LIN {X 0,Y 368.084,Z 680.12,A -85,B 0,C 180,E1 -13030.841,E2 -13030.841} C_VEL
LIN {X 0,Y 367.442,Z 693.726,A -85,B 0,C 180,E1 -13031.349,E2 -13031.349} C_VEL
LIN {X 0,Y 366.551,Z 706.591,A -85,B 0,C 180,E1 -13032.062,E2 -13032.062} C_VEL
LIN {X 0,Y 365.621,Z 718.366,A -85,B 0,C 180,E1 -13032.953,E2 -13032.953} C_VEL
LIN {X 0,Y 364.601,Z 729.747,A -85,B 0,C 180,E1 -13034.055,E2 -13034.055} C_VEL
LIN {X 0,Y 363.698,Z 740.032,A -85,B 0,C 180,E1 -13035.309,E2 -13035.309} C_VEL
LIN {X 0,Y 362.713,Z 750.07,A -85,B 0,C 180,E1 -13036.839,E2 -13036.839} C_VEL
LIN {X 0,Y 361.776,Z 758.914,A -85,B 0,C 180,E1 -13038.513,E2 -13038.513} C_VEL
LIN {X 0,Y 361.167,Z 765.962,A -85,B 0,C 180,E1 -13040.195,E2 -13040.195} C_VEL
LIN {X 0,Y 360.675,Z 772.412,A -85,B 0,C 180,E1 -13042.159,E2 -13042.159} C_VEL
LIN {X 0,Y 360.43,Z 776.906,A -85,B 0,C 180,E1 -13043.963,E2 -13043.963} C_VEL
LIN {X 0,Y 360.371,Z 779.772,A -85,B 0,C 180,E1 -13045.524,E2 -13045.524} C_VEL
LIN {X 0,Y 360.303,Z 781.326,A -85,B 0,C 180,E1 -13046.644,E2 -13046.644} C_VEL
LIN {X 0,Y 360.267,Z 782.42,A -85,B 0,C 180,E1 -13047.762,E2 -13047.762} C_VEL
LIN {X 0,Y 360.319,Z 783.103,A -85,B 0,C 180,E1 -13048.881,E2 -13048.881} C_VEL
LIN {X 0,Y 360.36,Z 783.39,A -85,B 0,C 180,E1 -13049.998,E2 -13049.998} C_VEL
LIN {X 0,Y 360.303,Z 783.278,A -85,B 0,C 180,E1 -13051.116,E2 -13051.116} C_VEL
LIN {X 0,Y 360.264,Z 782.727,A -85,B 0,C 180,E1 -13052.234,E2 -13052.234} C_VEL
LIN {X 0,Y 360.301,Z 781.769,A -85,B 0,C 180,E1 -13053.353,E2 -13053.353} C_VEL
LIN {X 0,Y 360.368,Z 780.41,A -85,B 0,C 180,E1 -13054.472,E2 -13054.472} C_VEL
LIN {X 0,Y 360.378,Z 777.924,A -85,B 0,C 180,E1 -13055.959,E2 -13055.959} C_VEL
LIN {X 0,Y 360.68,Z 773.636,A -85,B 0,C 180,E1 -13057.838,E2 -13057.838} C_VEL
LIN {X 0,Y 361.116,Z 768.601,A -85,B 0,C 180,E1 -13059.52,E2 -13059.52} C_VEL
LIN {X 0,Y 361.712,Z 762.283,A -85,B 0,C 180,E1 -13061.202,E2 -13061.202} C_VEL
LIN {X 0,Y 362.686,Z 754.4,A -85,B 0,C 180,E1 -13062.874,E2 -13062.874} C_VEL
LIN {X 0,Y 363.619,Z 746.365,A -85,B 0,C 180,E1 -13064.265,E2 -13064.265} C_VEL
LIN {X 0,Y 364.64,Z 736.582,A -85,B 0,C 180,E1 -13065.653,E2 -13065.653} C_VEL
LIN {X 0,Y 365.815,Z 725.732,A -85,B 0,C 180,E1 -13066.891,E2 -13066.891} C_VEL
LIN {X 0,Y 366.852,Z 715.177,A -85,B 0,C 180,E1 -13067.848,E2 -13067.848} C_VEL
LIN {X 0,Y 367.922,Z 702.54,A -85,B 0,C 180,E1 -13068.731,E2 -13068.731} C_VEL
LIN {X 0,Y 368.816,Z 690.014,A -85,B 0,C 180,E1 -13069.369,E2 -13069.369} C_VEL
LIN {X 0,Y 369.448,Z 677.021,A -85,B 0,C 180,E1 -13069.805,E2 -13069.805} C_VEL
LIN {X 0,Y 370.879,Z 603.724,A -85,B 0,C 180,E1 -13071.351,E2 -13071.351} C_VEL
LIN {X 0,Y 367.392,Z 581.766,A -85,B 0,C 180,E1 -13072.093,E2 -13072.093} C_VEL
LIN {X 0,Y 365.082,Z 570.344,A -85,B 0,C 180,E1 -13072.547,E2 -13072.547} C_VEL
LIN {X 0,Y 366.093,Z 561.386,A -85,B 0,C 180,E1 -13074.677,E2 -13074.677} C_VEL
LIN {X 0,Y 365.722,Z 557.159,A -85,B 0,C 180,E1 -13075.762,E2 -13075.762} C_VEL
LIN {X 0,Y 363.389,Z 545.667,A -85,B 0,C 180,E1 -13078.912,E2 -13078.912} C_VEL
LIN {X 0,Y 361.905,Z 539.407,A -85,B 0,C 180,E1 -13080.781,E2 -13080.781} C_VEL
LIN {X 0,Y 361.851,Z 539.411,A -85,B 0,C 180,E1 -13084.279,E2 -13084.279} C_VEL
LIN {X 0,Y 361.868,Z 539.412,A -85,B 0,C 180,E1 -13087.223,E2 -13087.223} C_VEL
LIN {X 0,Y 361.868,Z 539.412,A -85,B 0,C 180,E1 -13090.761,E2 -13090.761} C_VEL
LIN {X 0,Y 361.817,Z 539.417,A -85,B 0,C 180,E1 -13094.366,E2 -13094.366} C_VEL
LIN {X 0,Y 361.85,Z 539.412,A -85,B 0,C 180,E1 -13097.563,E2 -13097.563} C_VEL
LIN {X 0,Y 361.868,Z 539.408,A -85,B 0,C 180,E1 -13100.971,E2 -13100.971} C_VEL
LIN {X 0,Y 361.867,Z 539.408,A -85,B 0,C 180,E1 -13104.654,E2 -13104.654} C_VEL
LIN {X 0,Y 361.829,Z 539.41,A -85,B 0,C 180,E1 -13108.369,E2 -13108.369} C_VEL
LIN {X 0,Y 361.893,Z 539.406,A -85,B 0,C 180,E1 -13110.954,E2 -13110.954} C_VEL
LIN {X 0,Y 361.945,Z 539.396,A -85,B 0,C 180,E1 -13113.474,E2 -13113.474} C_VEL
LIN {X 0,Y 361.88,Z 539.401,A -85,B 0,C 180,E1 -13117.143,E2 -13117.143} C_VEL
LIN {X 0,Y 361.91,Z 539.394,A -85,B 0,C 180,E1 -13120.723,E2 -13120.723} C_VEL
LIN {X 0,Y 361.936,Z 539.392,A -85,B 0,C 180,E1 -13124.225,E2 -13124.225} C_VEL
LIN {X 0,Y 361.989,Z 539.392,A -85,B 0,C 180,E1 -13126.527,E2 -13126.527} C_VEL
LIN {X 0,Y 362.025,Z 539.389,A -85,B 0,C 180,E1 -13129.937,E2 -13129.937} C_VEL
LIN {X 0,Y 362.14,Z 539.37,A -85,B 0,C 180,E1 -13132.192,E2 -13132.192} C_VEL
LIN {X 0,Y 362.108,Z 539.376,A -85,B 0,C 180,E1 -13134.431,E2 -13134.431} C_VEL
LIN {X 0,Y 362.272,Z 539.356,A -85,B 0,C 180,E1 -13137.776,E2 -13137.776} C_VEL
LIN {X 0,Y 362.418,Z 539.341,A -85,B 0,C 180,E1 -13139.999,E2 -13139.999} C_VEL
LIN {X 0,Y 362.272,Z 539.356,A -85,B 0,C 180,E1 -13142.223,E2 -13142.223} C_VEL
LIN {X 0,Y 362.165,Z 539.372,A -85,B 0,C 180,E1 -13146.686,E2 -13146.686} C_VEL
LIN {X 0,Y 362.063,Z 539.386,A -85,B 0,C 180,E1 -13148.933,E2 -13148.933} C_VEL
LIN {X 0,Y 361.956,Z 539.398,A -85,B 0,C 180,E1 -13152.332,E2 -13152.332} C_VEL
LIN {X 0,Y 361.95,Z 539.401,A -85,B 0,C 180,E1 -13154.62,E2 -13154.62} C_VEL
LIN {X 0,Y 361.943,Z 539.402,A -85,B 0,C 180,E1 -13158.099,E2 -13158.099} C_VEL
LIN {X 0,Y 361.87,Z 539.407,A -85,B 0,C 180,E1 -13161.654,E2 -13161.654} C_VEL
LIN {X 0,Y 361.912,Z 539.488,A -85,B 0,C 180,E1 -13163.307,E2 -13163.307} C_VEL
LIN {X 0,Y 363.986,Z 549.132,A -85,B 0,C 180,E1 -13166.365,E2 -13166.365} C_VEL
LIN {X 0,Y 364.74,Z 552.95,A -85,B 0,C 180,E1 -13167.518,E2 -13167.518} C_VEL
LIN {X 0,Y 367.86,Z 561.593,A -85,B 0,C 180,E1 -13167.947,E2 -13167.947} C_VEL
LIN {X 0,Y 371.419,Z 578.984,A -85,B 0,C 180,E1 -13168.598,E2 -13168.598} C_VEL
LIN {X 0,Y 369.528,Z 660.348,A -85,B 0,C 180,E1 -13170.323,E2 -13170.323} C_VEL
LIN {X 0,Y 368.94,Z 673.355,A -85,B 0,C 180,E1 -13170.816,E2 -13170.816} C_VEL
LIN {X 0,Y 368.184,Z 685.745,A -85,B 0,C 180,E1 -13171.502,E2 -13171.502} C_VEL
LIN {X 0,Y 367.176,Z 697.789,A -85,B 0,C 180,E1 -13172.407,E2 -13172.407} C_VEL
LIN {X 0,Y 366.109,Z 709.182,A -85,B 0,C 180,E1 -13173.514,E2 -13173.514} C_VEL
LIN {X 0,Y 365.054,Z 719.145,A -85,B 0,C 180,E1 -13174.722,E2 -13174.722} C_VEL
LIN {X 0,Y 364.055,Z 727.868,A -85,B 0,C 180,E1 -13176.021,E2 -13176.021} C_VEL
LIN {X 0,Y 363.091,Z 735.885,A -85,B 0,C 180,E1 -13177.48,E2 -13177.48} C_VEL
LIN {X 0,Y 362.237,Z 743.126,A -85,B 0,C 180,E1 -13179.101,E2 -13179.101} C_VEL
LIN {X 0,Y 361.466,Z 749.878,A -85,B 0,C 180,E1 -13181.006,E2 -13181.006} C_VEL
LIN {X 0,Y 360.921,Z 755.115,A -85,B 0,C 180,E1 -13182.963,E2 -13182.963} C_VEL
LIN {X 0,Y 360.596,Z 758.312,A -85,B 0,C 180,E1 -13184.558,E2 -13184.558} C_VEL
LIN {X 0,Y 360.329,Z 760.647,A -85,B 0,C 180,E1 -13186.191,E2 -13186.191} C_VEL
LIN {X 0,Y 360.116,Z 762.378,A -85,B 0,C 180,E1 -13188.432,E2 -13188.432} C_VEL
LIN {X 0,Y 360.063,Z 762.667,A -85,B 0,C 180,E1 -13189.903,E2 -13189.903} C_VEL
LIN {X 0,Y 360.083,Z 762.241,A -85,B 0,C 180,E1 -13191.352,E2 -13191.352} C_VEL
LIN {X 0,Y 360.207,Z 760.809,A -85,B 0,C 180,E1 -13193.124,E2 -13193.124} C_VEL
LIN {X 0,Y 360.484,Z 758.216,A -85,B 0,C 180,E1 -13194.967,E2 -13194.967} C_VEL
LIN {X 0,Y 360.765,Z 754.078,A -85,B 0,C 180,E1 -13196.946,E2 -13196.946} C_VEL
LIN {X 0,Y 361.249,Z 748.549,A -85,B 0,C 180,E1 -13198.87,E2 -13198.87} C_VEL
LIN {X 0,Y 361.869,Z 742.009,A -85,B 0,C 180,E1 -13200.637,E2 -13200.637} C_VEL
LIN {X 0,Y 362.646,Z 734.341,A -85,B 0,C 180,E1 -13202.284,E2 -13202.284} C_VEL
LIN {X 0,Y 363.571,Z 724.85,A -85,B 0,C 180,E1 -13203.913,E2 -13203.913} C_VEL
LIN {X 0,Y 364.526,Z 714.942,A -85,B 0,C 180,E1 -13205.284,E2 -13205.284} C_VEL
LIN {X 0,Y 365.51,Z 704.514,A -85,B 0,C 180,E1 -13206.439,E2 -13206.439} C_VEL
LIN {X 0,Y 366.396,Z 693.123,A -85,B 0,C 180,E1 -13207.443,E2 -13207.443} C_VEL
LIN {X 0,Y 367.292,Z 680.176,A -85,B 0,C 180,E1 -13208.315,E2 -13208.315} C_VEL
LIN {X 0,Y 367.937,Z 667.003,A -85,B 0,C 180,E1 -13208.937,E2 -13208.937} C_VEL
LIN {X 0,Y 368.372,Z 653.798,A -85,B 0,C 180,E1 -13209.333,E2 -13209.333} C_VEL
LIN {X 0,Y 369.729,Z 577.273,A -85,B 0,C 180,E1 -13210.906,E2 -13210.906} C_VEL
LIN {X 0,Y 365.138,Z 554.624,A -85,B 0,C 180,E1 -13211.653,E2 -13211.653} C_VEL
LIN {X 0,Y 364.298,Z 551.805,A -85,B 0,C 180,E1 -13211.782,E2 -13211.782} C_VEL
LIN {X 0,Y 362.153,Z 540.301,A -85,B 0,C 180,E1 -13215.102,E2 -13215.102} C_VEL
LIN {X 0,Y 361.997,Z 539.395,A -85,B 0,C 180,E1 -13215.383,E2 -13215.383} C_VEL
LIN {X 0,Y 361.966,Z 539.4,A -85,B 0,C 180,E1 -13218.806,E2 -13218.806} C_VEL
LIN {X 0,Y 362.118,Z 539.375,A -85,B 0,C 180,E1 -13222.194,E2 -13222.194} C_VEL
LIN {X 0,Y 362.111,Z 539.377,A -85,B 0,C 180,E1 -13224.433,E2 -13224.433} C_VEL
LIN {X 0,Y 362.28,Z 539.354,A -85,B 0,C 180,E1 -13227.778,E2 -13227.778} C_VEL
LIN {X 0,Y 362.425,Z 539.336,A -85,B 0,C 180,E1 -13230.002,E2 -13230.002} C_VEL
LIN {X 0,Y 362.28,Z 539.354,A -85,B 0,C 180,E1 -13232.225,E2 -13232.225} C_VEL
LIN {X 0,Y 362.159,Z 539.372,A -85,B 0,C 180,E1 -13236.688,E2 -13236.688} C_VEL
LIN {X 0,Y 362.103,Z 539.378,A -85,B 0,C 180,E1 -13238.513,E2 -13238.513} C_VEL
LIN {X 0,Y 361.349,Z 539.476,A -85,B 0,C 180,E1 -13239.441,E2 -13239.441} C_VEL
LIN {X 0,Y 358.415,Z 539.841,A -85,B 0,C 180,E1 -13240.948,E2 -13240.948} C_VEL
LIN {X 0,Y 355.996,Z 540.137,A -85,B 0,C 180,E1 -13242.167,E2 -13242.167} C_VEL
LIN {X 0,Y 354.993,Z 540.268,A -85,B 0,C 180,E1 -13243.112,E2 -13243.112} C_VEL
LIN {X 0,Y 354.927,Z 540.269,A -85,B 0,C 180,E1 -13243.431,E2 -13243.431} C_VEL
LIN {X 0,Y 354.898,Z 540.278,A -85,B 0,C 180,E1 -13247.282,E2 -13247.282} C_VEL
LIN {X 0,Y 354.84,Z 540.285,A -85,B 0,C 180,E1 -13250.888,E2 -13250.888} C_VEL
LIN {X 0,Y 354.862,Z 540.279,A -85,B 0,C 180,E1 -13254.578,E2 -13254.578} C_VEL
LIN {X 0,Y 354.882,Z 540.281,A -85,B 0,C 180,E1 -13257.098,E2 -13257.098} C_VEL
LIN {X 0,Y 354.801,Z 540.29,A -85,B 0,C 180,E1 -13261,E2 -13261} C_VEL
LIN {X 0,Y 354.808,Z 540.287,A -85,B 0,C 180,E1 -13263.703,E2 -13263.703} C_VEL
LIN {X 0,Y 354.799,Z 540.286,A -85,B 0,C 180,E1 -13266.461,E2 -13266.461} C_VEL
LIN {X 0,Y 354.826,Z 540.288,A -85,B 0,C 180,E1 -13269.425,E2 -13269.425} C_VEL
LIN {X 0,Y 354.792,Z 540.289,A -85,B 0,C 180,E1 -13272.869,E2 -13272.869} C_VEL
LIN {X 0,Y 354.784,Z 540.288,A -85,B 0,C 180,E1 -13276.107,E2 -13276.107} C_VEL
LIN {X 0,Y 354.791,Z 540.291,A -85,B 0,C 180,E1 -13279.18,E2 -13279.18} C_VEL
LIN {X 0,Y 354.811,Z 540.284,A -85,B 0,C 180,E1 -13282.404,E2 -13282.404} C_VEL
LIN {X 0,Y 354.816,Z 540.285,A -85,B 0,C 180,E1 -13284.942,E2 -13284.942} C_VEL
LIN {X 0,Y 354.797,Z 540.286,A -85,B 0,C 180,E1 -13288.406,E2 -13288.406} C_VEL
LIN {X 0,Y 354.856,Z 540.285,A -85,B 0,C 180,E1 -13291.62,E2 -13291.62} C_VEL
LIN {X 0,Y 354.904,Z 540.274,A -85,B 0,C 180,E1 -13294.174,E2 -13294.174} C_VEL
LIN {X 0,Y 354.823,Z 540.286,A -85,B 0,C 180,E1 -13297.894,E2 -13297.894} C_VEL
LIN {X 0,Y 354.896,Z 540.277,A -85,B 0,C 180,E1 -13301.909,E2 -13301.909} C_VEL
LIN {X 0,Y 354.949,Z 540.271,A -85,B 0,C 180,E1 -13305.982,E2 -13305.982} C_VEL
LIN {X 0,Y 354.984,Z 540.269,A -85,B 0,C 180,E1 -13309.737,E2 -13309.737} C_VEL
LIN {X 0,Y 355.132,Z 540.246,A -85,B 0,C 180,E1 -13313.181,E2 -13313.181} C_VEL
LIN {X 0,Y 355.251,Z 540.235,A -85,B 0,C 180,E1 -13317.733,E2 -13317.733} C_VEL
LIN {X 0,Y 355.403,Z 540.215,A -85,B 0,C 180,E1 -13320.001,E2 -13320.001} C_VEL
LIN {X 0,Y 355.251,Z 540.232,A -85,B 0,C 180,E1 -13322.268,E2 -13322.268} C_VEL
LIN {X 0,Y 355.146,Z 540.243,A -85,B 0,C 180,E1 -13326.82,E2 -13326.82} C_VEL
LIN {X 0,Y 355.023,Z 540.258,A -85,B 0,C 180,E1 -13329.113,E2 -13329.113} C_VEL
LIN {X 0,Y 354.929,Z 540.271,A -85,B 0,C 180,E1 -13332.581,E2 -13332.581} C_VEL
LIN {X 0,Y 354.898,Z 540.279,A -85,B 0,C 180,E1 -13336.096,E2 -13336.096} C_VEL
LIN {X 0,Y 354.912,Z 540.274,A -85,B 0,C 180,E1 -13338.472,E2 -13338.472} C_VEL
LIN {X 0,Y 354.824,Z 540.289,A -85,B 0,C 180,E1 -13342.107,E2 -13342.107} C_VEL
LIN {X 0,Y 354.906,Z 540.276,A -85,B 0,C 180,E1 -13345.827,E2 -13345.827} C_VEL
LIN {X 0,Y 354.826,Z 540.285,A -85,B 0,C 180,E1 -13349.682,E2 -13349.682} C_VEL
LIN {X 0,Y 354.814,Z 540.286,A -85,B 0,C 180,E1 -13353.702,E2 -13353.702} C_VEL
LIN {X 0,Y 354.806,Z 540.289,A -85,B 0,C 180,E1 -13356.459,E2 -13356.459} C_VEL
LIN {X 0,Y 354.832,Z 540.282,A -85,B 0,C 180,E1 -13359.423,E2 -13359.423} C_VEL
LIN {X 0,Y 354.795,Z 540.287,A -85,B 0,C 180,E1 -13362.867,E2 -13362.867} C_VEL
LIN {X 0,Y 354.775,Z 540.293,A -85,B 0,C 180,E1 -13366.103,E2 -13366.103} C_VEL
LIN {X 0,Y 354.796,Z 540.286,A -85,B 0,C 180,E1 -13369.178,E2 -13369.178} C_VEL
LIN {X 0,Y 354.82,Z 540.289,A -85,B 0,C 180,E1 -13372.401,E2 -13372.401} C_VEL
LIN {X 0,Y 354.819,Z 540.285,A -85,B 0,C 180,E1 -13374.94,E2 -13374.94} C_VEL
LIN {X 0,Y 354.801,Z 540.292,A -85,B 0,C 180,E1 -13378.404,E2 -13378.404} C_VEL
LIN {X 0,Y 354.856,Z 540.352,A -85,B 0,C 180,E1 -13380.034,E2 -13380.034} C_VEL
LIN {X 0,Y 357.26,Z 551.762,A -85,B 0,C 180,E1 -13383.097,E2 -13383.097} C_VEL
LIN {X 0,Y 358.602,Z 559.43,A -85,B 0,C 180,E1 -13385.078,E2 -13385.078} C_VEL
LIN {X 0,Y 357.874,Z 568.426,A -85,B 0,C 180,E1 -13387.225,E2 -13387.225} C_VEL
LIN {X 0,Y 357.564,Z 571.17,A -85,B 0,C 180,E1 -13387.87,E2 -13387.87} C_VEL
LIN {X 0,Y 362.726,Z 604.121,A -85,B 0,C 180,E1 -13388.896,E2 -13388.896} C_VEL
LIN {X 0,Y 361.331,Z 679.629,A -85,B 0,C 180,E1 -13390.505,E2 -13390.505} C_VEL
LIN {X 0,Y 360.654,Z 693.32,A -85,B 0,C 180,E1 -13391.022,E2 -13391.022} C_VEL
LIN {X 0,Y 359.796,Z 705.738,A -85,B 0,C 180,E1 -13391.713,E2 -13391.713} C_VEL
LIN {X 0,Y 358.808,Z 717.665,A -85,B 0,C 180,E1 -13392.619,E2 -13392.619} C_VEL
LIN {X 0,Y 357.724,Z 729.14,A -85,B 0,C 180,E1 -13393.741,E2 -13393.741} C_VEL
LIN {X 0,Y 356.804,Z 739.453,A -85,B 0,C 180,E1 -13395.008,E2 -13395.008} C_VEL
LIN {X 0,Y 355.739,Z 749.626,A -85,B 0,C 180,E1 -13396.576,E2 -13396.576} C_VEL
LIN {X 0,Y 354.759,Z 758.519,A -85,B 0,C 180,E1 -13398.283,E2 -13398.283} C_VEL
LIN {X 0,Y 354.129,Z 765.615,A -85,B 0,C 180,E1 -13399.998,E2 -13399.998} C_VEL
LIN {X 0,Y 353.619,Z 772.097,A -85,B 0,C 180,E1 -13402.001,E2 -13402.001} C_VEL
LIN {X 0,Y 353.324,Z 777.005,A -85,B 0,C 180,E1 -13404.022,E2 -13404.022} C_VEL
LIN {X 0,Y 353.284,Z 779.509,A -85,B 0,C 180,E1 -13405.434,E2 -13405.434} C_VEL
LIN {X 0,Y 353.225,Z 781.075,A -85,B 0,C 180,E1 -13406.576,E2 -13406.576} C_VEL
LIN {X 0,Y 353.175,Z 782.189,A -85,B 0,C 180,E1 -13407.717,E2 -13407.717} C_VEL
LIN {X 0,Y 353.219,Z 782.882,A -85,B 0,C 180,E1 -13408.858,E2 -13408.858} C_VEL
LIN {X 0,Y 353.263,Z 783.178,A -85,B 0,C 180,E1 -13409.998,E2 -13409.998} C_VEL
LIN {X 0,Y 353.204,Z 783.078,A -85,B 0,C 180,E1 -13411.139,E2 -13411.139} C_VEL
LIN {X 0,Y 353.173,Z 782.544,A -85,B 0,C 180,E1 -13412.279,E2 -13412.279} C_VEL
LIN {X 0,Y 353.223,Z 781.596,A -85,B 0,C 180,E1 -13413.42,E2 -13413.42} C_VEL
LIN {X 0,Y 353.281,Z 780.249,A -85,B 0,C 180,E1 -13414.562,E2 -13414.562} C_VEL
LIN {X 0,Y 353.297,Z 778.061,A -85,B 0,C 180,E1 -13415.935,E2 -13415.935} C_VEL
LIN {X 0,Y 353.624,Z 773.526,A -85,B 0,C 180,E1 -13417.995,E2 -13417.995} C_VEL
LIN {X 0,Y 354.076,Z 768.515,A -85,B 0,C 180,E1 -13419.711,E2 -13419.711} C_VEL
LIN {X 0,Y 354.713,Z 762.222,A -85,B 0,C 180,E1 -13421.426,E2 -13421.426} C_VEL
LIN {X 0,Y 355.741,Z 754.384,A -85,B 0,C 180,E1 -13423.13,E2 -13423.13} C_VEL
LIN {X 0,Y 356.705,Z 746.384,A -85,B 0,C 180,E1 -13424.547,E2 -13424.547} C_VEL
LIN {X 0,Y 357.795,Z 736.642,A -85,B 0,C 180,E1 -13425.96,E2 -13425.96} C_VEL
LIN {X 0,Y 359.026,Z 725.85,A -85,B 0,C 180,E1 -13427.22,E2 -13427.22} C_VEL
LIN {X 0,Y 360.124,Z 715.408,A -85,B 0,C 180,E1 -13428.193,E2 -13428.193} C_VEL
LIN {X 0,Y 361.232,Z 702.941,A -85,B 0,C 180,E1 -13429.091,E2 -13429.091} C_VEL
LIN {X 0,Y 362.16,Z 690.663,A -85,B 0,C 180,E1 -13429.74,E2 -13429.74} C_VEL
LIN {X 0,Y 362.801,Z 678.427,A -85,B 0,C 180,E1 -13430.183,E2 -13430.183} C_VEL
LIN {X 0,Y 364.355,Z 604.435,A -85,B 0,C 180,E1 -13431.787,E2 -13431.787} C_VEL
LIN {X 0,Y 360.878,Z 582.501,A -85,B 0,C 180,E1 -13432.549,E2 -13432.549} C_VEL
LIN {X 0,Y 358.355,Z 570.184,A -85,B 0,C 180,E1 -13433.044,E2 -13433.044} C_VEL
LIN {X 0,Y 359.237,Z 562.67,A -85,B 0,C 180,E1 -13434.872,E2 -13434.872} C_VEL
LIN {X 0,Y 358.671,Z 557.744,A -85,B 0,C 180,E1 -13436.179,E2 -13436.179} C_VEL
LIN {X 0,Y 356.453,Z 547.013,A -85,B 0,C 180,E1 -13439.206,E2 -13439.206} C_VEL
LIN {X 0,Y 354.812,Z 540.292,A -85,B 0,C 180,E1 -13441.269,E2 -13441.269} C_VEL
LIN {X 0,Y 354.809,Z 540.29,A -85,B 0,C 180,E1 -13445.057,E2 -13445.057} C_VEL
LIN {X 0,Y 354.807,Z 540.293,A -85,B 0,C 180,E1 -13447.88,E2 -13447.88} C_VEL
LIN {X 0,Y 354.812,Z 540.294,A -85,B 0,C 180,E1 -13451.175,E2 -13451.175} C_VEL
LIN {X 0,Y 354.784,Z 540.294,A -85,B 0,C 180,E1 -13454.509,E2 -13454.509} C_VEL
LIN {X 0,Y 354.807,Z 540.29,A -85,B 0,C 180,E1 -13457.664,E2 -13457.664} C_VEL
LIN {X 0,Y 354.83,Z 540.284,A -85,B 0,C 180,E1 -13460.667,E2 -13460.667} C_VEL
LIN {X 0,Y 354.815,Z 540.287,A -85,B 0,C 180,E1 -13464.299,E2 -13464.299} C_VEL
LIN {X 0,Y 354.779,Z 540.293,A -85,B 0,C 180,E1 -13467.665,E2 -13467.665} C_VEL
LIN {X 0,Y 354.86,Z 540.28,A -85,B 0,C 180,E1 -13470.62,E2 -13470.62} C_VEL
LIN {X 0,Y 354.89,Z 540.277,A -85,B 0,C 180,E1 -13474.171,E2 -13474.171} C_VEL
LIN {X 0,Y 354.825,Z 540.287,A -85,B 0,C 180,E1 -13477.893,E2 -13477.893} C_VEL
LIN {X 0,Y 354.913,Z 540.276,A -85,B 0,C 180,E1 -13481.89,E2 -13481.89} C_VEL
LIN {X 0,Y 354.933,Z 540.273,A -85,B 0,C 180,E1 -13485.98,E2 -13485.98} C_VEL
LIN {X 0,Y 354.972,Z 540.27,A -85,B 0,C 180,E1 -13489.735,E2 -13489.735} C_VEL
LIN {X 0,Y 355.103,Z 540.246,A -85,B 0,C 180,E1 -13492.036,E2 -13492.036} C_VEL
LIN {X 0,Y 355.082,Z 540.252,A -85,B 0,C 180,E1 -13494.32,E2 -13494.32} C_VEL
LIN {X 0,Y 355.235,Z 540.233,A -85,B 0,C 180,E1 -13497.732,E2 -13497.732} C_VEL
LIN {X 0,Y 355.388,Z 540.217,A -85,B 0,C 180,E1 -13499.999,E2 -13499.999} C_VEL
LIN {X 0,Y 355.235,Z 540.232,A -85,B 0,C 180,E1 -13502.267,E2 -13502.267} C_VEL
LIN {X 0,Y 355.13,Z 540.249,A -85,B 0,C 180,E1 -13506.819,E2 -13506.819} C_VEL
LIN {X 0,Y 355.005,Z 540.266,A -85,B 0,C 180,E1 -13509.112,E2 -13509.112} C_VEL
LIN {X 0,Y 354.915,Z 540.276,A -85,B 0,C 180,E1 -13512.58,E2 -13512.58} C_VEL
LIN {X 0,Y 354.878,Z 540.284,A -85,B 0,C 180,E1 -13516.096,E2 -13516.096} C_VEL
LIN {X 0,Y 354.889,Z 540.28,A -85,B 0,C 180,E1 -13518.472,E2 -13518.472} C_VEL
LIN {X 0,Y 354.818,Z 540.288,A -85,B 0,C 180,E1 -13522.106,E2 -13522.106} C_VEL
LIN {X 0,Y 354.86,Z 540.479,A -85,B 0,C 180,E1 -13522.871,E2 -13522.871} C_VEL
LIN {X 0,Y 357.157,Z 550.944,A -85,B 0,C 180,E1 -13526.279,E2 -13526.279} C_VEL
LIN {X 0,Y 357.576,Z 553.097,A -85,B 0,C 180,E1 -13526.954,E2 -13526.954} C_VEL
LIN {X 0,Y 361.632,Z 563.76,A -85,B 0,C 180,E1 -13527.539,E2 -13527.539} C_VEL
LIN {X 0,Y 364.939,Z 579.586,A -85,B 0,C 180,E1 -13528.152,E2 -13528.152} C_VEL
LIN {X 0,Y 362.969,Z 660.454,A -85,B 0,C 180,E1 -13529.901,E2 -13529.901} C_VEL
LIN {X 0,Y 362.332,Z 673.727,A -85,B 0,C 180,E1 -13530.413,E2 -13530.413} C_VEL
LIN {X 0,Y 361.622,Z 685.296,A -85,B 0,C 180,E1 -13531.066,E2 -13531.066} C_VEL
LIN {X 0,Y 360.636,Z 696.671,A -85,B 0,C 180,E1 -13531.911,E2 -13531.911} C_VEL
LIN {X 0,Y 359.463,Z 708.748,A -85,B 0,C 180,E1 -13533.087,E2 -13533.087} C_VEL
LIN {X 0,Y 358.248,Z 719.445,A -85,B 0,C 180,E1 -13534.398,E2 -13534.398} C_VEL
LIN {X 0,Y 357.137,Z 728.637,A -85,B 0,C 180,E1 -13535.805,E2 -13535.805} C_VEL
LIN {X 0,Y 356.083,Z 736.914,A -85,B 0,C 180,E1 -13537.366,E2 -13537.366} C_VEL
LIN {X 0,Y 355.26,Z 743.586,A -85,B 0,C 180,E1 -13538.909,E2 -13538.909} C_VEL
LIN {X 0,Y 354.433,Z 750.351,A -85,B 0,C 180,E1 -13540.87,E2 -13540.87} C_VEL
LIN {X 0,Y 353.897,Z 755.184,A -85,B 0,C 180,E1 -13542.714,E2 -13542.714} C_VEL
LIN {X 0,Y 353.57,Z 758.367,A -85,B 0,C 180,E1 -13544.312,E2 -13544.312} C_VEL
LIN {X 0,Y 353.288,Z 760.61,A -85,B 0,C 180,E1 -13545.875,E2 -13545.875} C_VEL
LIN {X 0,Y 353.104,Z 762.068,A -85,B 0,C 180,E1 -13547.427,E2 -13547.427} C_VEL
LIN {X 0,Y 352.986,Z 762.819,A -85,B 0,C 180,E1 -13549.163,E2 -13549.163} C_VEL
LIN {X 0,Y 352.958,Z 762.622,A -85,B 0,C 180,E1 -13550.945,E2 -13550.945} C_VEL
LIN {X 0,Y 353.073,Z 761.396,A -85,B 0,C 180,E1 -13552.769,E2 -13552.769} C_VEL
LIN {X 0,Y 353.348,Z 758.817,A -85,B 0,C 180,E1 -13554.776,E2 -13554.776} C_VEL
LIN {X 0,Y 353.592,Z 755.322,A -85,B 0,C 180,E1 -13556.593,E2 -13556.593} C_VEL
LIN {X 0,Y 354.088,Z 750.076,A -85,B 0,C 180,E1 -13558.59,E2 -13558.59} C_VEL
LIN {X 0,Y 354.649,Z 744.189,A -85,B 0,C 180,E1 -13560.305,E2 -13560.305} C_VEL
LIN {X 0,Y 355.411,Z 737.131,A -85,B 0,C 180,E1 -13561.951,E2 -13561.951} C_VEL
LIN {X 0,Y 356.335,Z 728.057,A -85,B 0,C 180,E1 -13563.657,E2 -13563.657} C_VEL
LIN {X 0,Y 357.283,Z 718.46,A -85,B 0,C 180,E1 -13565.103,E2 -13565.103} C_VEL
LIN {X 0,Y 358.461,Z 707.149,A -85,B 0,C 180,E1 -13566.457,E2 -13566.457} C_VEL
LIN {X 0,Y 359.328,Z 697.009,A -85,B 0,C 180,E1 -13567.43,E2 -13567.43} C_VEL
LIN {X 0,Y 360.085,Z 686.521,A -85,B 0,C 180,E1 -13568.235,E2 -13568.235} C_VEL
LIN {X 0,Y 360.807,Z 674.071,A -85,B 0,C 180,E1 -13568.958,E2 -13568.958} C_VEL
LIN {X 0,Y 361.361,Z 660.996,A -85,B 0,C 180,E1 -13569.475,E2 -13569.475} C_VEL
LIN {X 0,Y 361.907,Z 635.849,A -85,B 0,C 180,E1 -13570.042,E2 -13570.042} C_VEL
LIN {X 0,Y 363.072,Z 579.027,A -85,B 0,C 180,E1 -13571.229,E2 -13571.229} C_VEL
LIN {X 0,Y 358.708,Z 556.769,A -85,B 0,C 180,E1 -13571.973,E2 -13571.973} C_VEL
LIN {X 0,Y 357.124,Z 551.949,A -85,B 0,C 180,E1 -13572.205,E2 -13572.205} C_VEL
LIN {X 0,Y 354.959,Z 540.27,A -85,B 0,C 180,E1 -13575.678,E2 -13575.678} C_VEL
LIN {X 0,Y 354.973,Z 540.264,A -85,B 0,C 180,E1 -13579.737,E2 -13579.737} C_VEL
LIN {X 0,Y 355.121,Z 540.249,A -85,B 0,C 180,E1 -13583.182,E2 -13583.182} C_VEL
LIN {X 0,Y 355.243,Z 540.231,A -85,B 0,C 180,E1 -13587.734,E2 -13587.734} C_VEL
LIN {X 0,Y 355.395,Z 540.212,A -85,B 0,C 180,E1 -13590.002,E2 -13590.002} C_VEL
LIN {X 0,Y 355.243,Z 540.231,A -85,B 0,C 180,E1 -13592.269,E2 -13592.269} C_VEL
LIN {X 0,Y 355.123,Z 540.25,A -85,B 0,C 180,E1 -13596.821,E2 -13596.821} C_VEL
LIN {X 0,Y 354.977,Z 540.264,A -85,B 0,C 180,E1 -13600.266,E2 -13600.266} C_VEL
LIN {X 0,Y 354.927,Z 540.269,A -85,B 0,C 180,E1 -13603.431,E2 -13603.431} C_VEL
LIN {X 0,Y 354.312,Z 540.349,A -85,B 0,C 180,E1 -13604.378,E2 -13604.378} C_VEL
LIN {X 0,Y 351.499,Z 540.697,A -85,B 0,C 180,E1 -13605.918,E2 -13605.918} C_VEL
LIN {X 0,Y 349.063,Z 541.006,A -85,B 0,C 180,E1 -13607.164,E2 -13607.164} C_VEL
LIN {X 0,Y 347.981,Z 541.136,A -85,B 0,C 180,E1 -13608.128,E2 -13608.128} C_VEL
LIN {X 0,Y 347.875,Z 541.149,A -85,B 0,C 180,E1 -13608.455,E2 -13608.455} C_VEL
LIN {X 0,Y 347.789,Z 541.161,A -85,B 0,C 180,E1 -13611.637,E2 -13611.637} C_VEL
LIN {X 0,Y 347.813,Z 541.162,A -85,B 0,C 180,E1 -13615.11,E2 -13615.11} C_VEL
LIN {X 0,Y 347.809,Z 541.158,A -85,B 0,C 180,E1 -13617.696,E2 -13617.696} C_VEL
LIN {X 0,Y 347.75,Z 541.164,A -85,B 0,C 180,E1 -13620.349,E2 -13620.349} C_VEL
LIN {X 0,Y 347.75,Z 541.164,A -85,B 0,C 180,E1 -13624.045,E2 -13624.045} C_VEL
LIN {X 0,Y 347.764,Z 541.169,A -85,B 0,C 180,E1 -13627.322,E2 -13627.322} C_VEL
LIN {X 0,Y 347.735,Z 541.166,A -85,B 0,C 180,E1 -13630.298,E2 -13630.298} C_VEL
LIN {X 0,Y 347.727,Z 541.173,A -85,B 0,C 180,E1 -13633.409,E2 -13633.409} C_VEL
LIN {X 0,Y 347.731,Z 541.167,A -85,B 0,C 180,E1 -13636.687,E2 -13636.687} C_VEL
LIN {X 0,Y 347.751,Z 541.164,A -85,B 0,C 180,E1 -13640.174,E2 -13640.174} C_VEL
LIN {X 0,Y 347.765,Z 541.162,A -85,B 0,C 180,E1 -13642.681,E2 -13642.681} C_VEL
LIN {X 0,Y 347.753,Z 541.166,A -85,B 0,C 180,E1 -13645.957,E2 -13645.957} C_VEL
LIN {X 0,Y 347.769,Z 541.167,A -85,B 0,C 180,E1 -13649.655,E2 -13649.655} C_VEL
LIN {X 0,Y 347.857,Z 541.151,A -85,B 0,C 180,E1 -13652.746,E2 -13652.746} C_VEL
LIN {X 0,Y 347.791,Z 541.16,A -85,B 0,C 180,E1 -13656.163,E2 -13656.163} C_VEL
LIN {X 0,Y 347.806,Z 541.16,A -85,B 0,C 180,E1 -13659.91,E2 -13659.91} C_VEL
LIN {X 0,Y 347.838,Z 541.158,A -85,B 0,C 180,E1 -13663.569,E2 -13663.569} C_VEL
LIN {X 0,Y 347.897,Z 541.147,A -85,B 0,C 180,E1 -13667.161,E2 -13667.161} C_VEL
LIN {X 0,Y 347.952,Z 541.139,A -85,B 0,C 180,E1 -13670.702,E2 -13670.702} C_VEL
LIN {X 0,Y 348.098,Z 541.121,A -85,B 0,C 180,E1 -13673.043,E2 -13673.043} C_VEL
LIN {X 0,Y 348.213,Z 541.112,A -85,B 0,C 180,E1 -13677.687,E2 -13677.687} C_VEL
LIN {X 0,Y 348.352,Z 541.094,A -85,B 0,C 180,E1 -13680.001,E2 -13680.001} C_VEL
LIN {X 0,Y 348.213,Z 541.108,A -85,B 0,C 180,E1 -13682.314,E2 -13682.314} C_VEL
LIN {X 0,Y 348.114,Z 541.119,A -85,B 0,C 180,E1 -13686.958,E2 -13686.958} C_VEL
LIN {X 0,Y 347.976,Z 541.137,A -85,B 0,C 180,E1 -13689.299,E2 -13689.299} C_VEL
LIN {X 0,Y 347.898,Z 541.146,A -85,B 0,C 180,E1 -13692.84,E2 -13692.84} C_VEL
LIN {X 0,Y 347.847,Z 541.154,A -85,B 0,C 180,E1 -13696.432,E2 -13696.432} C_VEL
LIN {X 0,Y 347.861,Z 541.15,A -85,B 0,C 180,E1 -13698.861,E2 -13698.861} C_VEL
LIN {X 0,Y 347.77,Z 541.163,A -85,B 0,C 180,E1 -13702.58,E2 -13702.58} C_VEL
LIN {X 0,Y 347.819,Z 541.155,A -85,B 0,C 180,E1 -13705.108,E2 -13705.108} C_VEL
LIN {X 0,Y 347.817,Z 541.158,A -85,B 0,C 180,E1 -13707.694,E2 -13707.694} C_VEL
LIN {X 0,Y 347.757,Z 541.167,A -85,B 0,C 180,E1 -13710.348,E2 -13710.348} C_VEL
LIN {X 0,Y 347.757,Z 541.168,A -85,B 0,C 180,E1 -13714.043,E2 -13714.043} C_VEL
LIN {X 0,Y 347.769,Z 541.162,A -85,B 0,C 180,E1 -13717.321,E2 -13717.321} C_VEL
LIN {X 0,Y 347.74,Z 541.171,A -85,B 0,C 180,E1 -13720.297,E2 -13720.297} C_VEL
LIN {X 0,Y 347.731,Z 541.166,A -85,B 0,C 180,E1 -13723.408,E2 -13723.408} C_VEL
LIN {X 0,Y 347.733,Z 541.169,A -85,B 0,C 180,E1 -13726.686,E2 -13726.686} C_VEL
LIN {X 0,Y 347.755,Z 541.168,A -85,B 0,C 180,E1 -13730.172,E2 -13730.172} C_VEL
LIN {X 0,Y 347.773,Z 541.164,A -85,B 0,C 180,E1 -13732.679,E2 -13732.679} C_VEL
LIN {X 0,Y 347.756,Z 541.165,A -85,B 0,C 180,E1 -13735.955,E2 -13735.955} C_VEL
LIN {X 0,Y 347.823,Z 541.195,A -85,B 0,C 180,E1 -13739.702,E2 -13739.702} C_VEL
LIN {X 0,Y 350.202,Z 552.602,A -85,B 0,C 180,E1 -13742.833,E2 -13742.833} C_VEL
LIN {X 0,Y 351.539,Z 559.674,A -85,B 0,C 180,E1 -13744.706,E2 -13744.706} C_VEL
LIN {X 0,Y 351.448,Z 564.074,A -85,B 0,C 180,E1 -13745.797,E2 -13745.797} C_VEL
LIN {X 0,Y 350.706,Z 570.943,A -85,B 0,C 180,E1 -13747.454,E2 -13747.454} C_VEL
LIN {X 0,Y 356.021,Z 605.298,A -85,B 0,C 180,E1 -13748.56,E2 -13748.56} C_VEL
LIN {X 0,Y 354.54,Z 680.037,A -85,B 0,C 180,E1 -13750.192,E2 -13750.192} C_VEL
LIN {X 0,Y 353.842,Z 693.523,A -85,B 0,C 180,E1 -13750.717,E2 -13750.717} C_VEL
LIN {X 0,Y 352.935,Z 705.813,A -85,B 0,C 180,E1 -13751.42,E2 -13751.42} C_VEL
LIN {X 0,Y 351.851,Z 718.467,A -85,B 0,C 180,E1 -13752.414,E2 -13752.414} C_VEL
LIN {X 0,Y 350.744,Z 729.762,A -85,B 0,C 180,E1 -13753.557,E2 -13753.557} C_VEL
LIN {X 0,Y 349.797,Z 739.944,A -85,B 0,C 180,E1 -13754.858,E2 -13754.858} C_VEL
LIN {X 0,Y 348.76,Z 749.122,A -85,B 0,C 180,E1 -13756.302,E2 -13756.302} C_VEL
LIN {X 0,Y 347.772,Z 758.072,A -85,B 0,C 180,E1 -13758.044,E2 -13758.044} C_VEL
LIN {X 0,Y 347.096,Z 765.235,A -85,B 0,C 180,E1 -13759.793,E2 -13759.793} C_VEL
LIN {X 0,Y 346.558,Z 771.756,A -85,B 0,C 180,E1 -13761.837,E2 -13761.837} C_VEL
LIN {X 0,Y 346.288,Z 776.04,A -85,B 0,C 180,E1 -13763.59,E2 -13763.59} C_VEL
LIN {X 0,Y 346.2,Z 779.232,A -85,B 0,C 180,E1 -13765.341,E2 -13765.341} C_VEL
LIN {X 0,Y 346.149,Z 780.813,A -85,B 0,C 180,E1 -13766.506,E2 -13766.506} C_VEL
LIN {X 0,Y 346.087,Z 781.952,A -85,B 0,C 180,E1 -13767.671,E2 -13767.671} C_VEL
LIN {X 0,Y 346.119,Z 782.657,A -85,B 0,C 180,E1 -13768.835,E2 -13768.835} C_VEL
LIN {X 0,Y 346.165,Z 782.966,A -85,B 0,C 180,E1 -13769.998,E2 -13769.998} C_VEL
LIN {X 0,Y 346.104,Z 782.877,A -85,B 0,C 180,E1 -13771.162,E2 -13771.162} C_VEL
LIN {X 0,Y 346.084,Z 782.367,A -85,B 0,C 180,E1 -13772.326,E2 -13772.326} C_VEL
LIN {X 0,Y 346.147,Z 781.431,A -85,B 0,C 180,E1 -13773.49,E2 -13773.49} C_VEL
LIN {X 0,Y 346.176,Z 780.093,A -85,B 0,C 180,E1 -13774.656,E2 -13774.656} C_VEL
LIN {X 0,Y 346.261,Z 777.273,A -85,B 0,C 180,E1 -13776.407,E2 -13776.407} C_VEL
LIN {X 0,Y 346.568,Z 773.416,A -85,B 0,C 180,E1 -13778.159,E2 -13778.159} C_VEL
LIN {X 0,Y 347.054,Z 768.428,A -85,B 0,C 180,E1 -13779.91,E2 -13779.91} C_VEL
LIN {X 0,Y 347.726,Z 762.16,A -85,B 0,C 180,E1 -13781.659,E2 -13781.659} C_VEL
LIN {X 0,Y 348.804,Z 754.368,A -85,B 0,C 180,E1 -13783.396,E2 -13783.396} C_VEL
LIN {X 0,Y 349.804,Z 746.421,A -85,B 0,C 180,E1 -13784.841,E2 -13784.841} C_VEL
LIN {X 0,Y 350.967,Z 736.75,A -85,B 0,C 180,E1 -13786.279,E2 -13786.279} C_VEL
LIN {X 0,Y 352.256,Z 726.047,A -85,B 0,C 180,E1 -13787.562,E2 -13787.562} C_VEL
LIN {X 0,Y 353.398,Z 715.731,A -85,B 0,C 180,E1 -13788.552,E2 -13788.552} C_VEL
LIN {X 0,Y 354.559,Z 703.462,A -85,B 0,C 180,E1 -13789.464,E2 -13789.464} C_VEL
LIN {X 0,Y 355.566,Z 690.692,A -85,B 0,C 180,E1 -13790.159,E2 -13790.159} C_VEL
LIN {X 0,Y 356.299,Z 677.39,A -85,B 0,C 180,E1 -13790.644,E2 -13790.644} C_VEL
LIN {X 0,Y 357.902,Z 605.372,A -85,B 0,C 180,E1 -13792.23,E2 -13792.23} C_VEL
LIN {X 0,Y 354.479,Z 583.806,A -85,B 0,C 180,E1 -13793.007,E2 -13793.007} C_VEL
LIN {X 0,Y 351.635,Z 569.896,A -85,B 0,C 180,E1 -13793.599,E2 -13793.599} C_VEL
LIN {X 0,Y 352.379,Z 563.973,A -85,B 0,C 180,E1 -13795.074,E2 -13795.074} C_VEL
LIN {X 0,Y 351.754,Z 559.131,A -85,B 0,C 180,E1 -13796.393,E2 -13796.393} C_VEL
LIN {X 0,Y 349.543,Z 548.516,A -85,B 0,C 180,E1 -13799.469,E2 -13799.469} C_VEL
LIN {X 0,Y 347.744,Z 541.173,A -85,B 0,C 180,E1 -13801.809,E2 -13801.809} C_VEL
LIN {X 0,Y 347.786,Z 541.165,A -85,B 0,C 180,E1 -13805.873,E2 -13805.873} C_VEL
LIN {X 0,Y 347.762,Z 541.169,A -85,B 0,C 180,E1 -13808.789,E2 -13808.789} C_VEL
LIN {X 0,Y 347.761,Z 541.172,A -85,B 0,C 180,E1 -13811.826,E2 -13811.826} C_VEL
LIN {X 0,Y 347.731,Z 541.172,A -85,B 0,C 180,E1 -13815.02,E2 -13815.02} C_VEL
LIN {X 0,Y 347.761,Z 541.167,A -85,B 0,C 180,E1 -13818.392,E2 -13818.392} C_VEL
LIN {X 0,Y 347.769,Z 541.162,A -85,B 0,C 180,E1 -13822.009,E2 -13822.009} C_VEL
LIN {X 0,Y 347.737,Z 541.165,A -85,B 0,C 180,E1 -13825.535,E2 -13825.535} C_VEL
LIN {X 0,Y 347.756,Z 541.163,A -85,B 0,C 180,E1 -13829.652,E2 -13829.652} C_VEL
LIN {X 0,Y 347.843,Z 541.149,A -85,B 0,C 180,E1 -13832.743,E2 -13832.743} C_VEL
LIN {X 0,Y 347.779,Z 541.156,A -85,B 0,C 180,E1 -13836.161,E2 -13836.161} C_VEL
LIN {X 0,Y 347.807,Z 541.152,A -85,B 0,C 180,E1 -13839.908,E2 -13839.908} C_VEL
LIN {X 0,Y 347.856,Z 541.153,A -85,B 0,C 180,E1 -13842.358,E2 -13842.358} C_VEL
LIN {X 0,Y 347.887,Z 541.151,A -85,B 0,C 180,E1 -13845.97,E2 -13845.97} C_VEL
LIN {X 0,Y 347.922,Z 541.147,A -85,B 0,C 180,E1 -13849.525,E2 -13849.525} C_VEL
LIN {X 0,Y 348.063,Z 541.123,A -85,B 0,C 180,E1 -13851.874,E2 -13851.874} C_VEL
LIN {X 0,Y 348.057,Z 541.127,A -85,B 0,C 180,E1 -13854.205,E2 -13854.205} C_VEL
LIN {X 0,Y 348.198,Z 541.11,A -85,B 0,C 180,E1 -13857.686,E2 -13857.686} C_VEL
LIN {X 0,Y 348.357,Z 541.092,A -85,B 0,C 180,E1 -13859.999,E2 -13859.999} C_VEL
LIN {X 0,Y 348.198,Z 541.109,A -85,B 0,C 180,E1 -13862.313,E2 -13862.313} C_VEL
LIN {X 0,Y 348.098,Z 541.124,A -85,B 0,C 180,E1 -13866.957,E2 -13866.957} C_VEL
LIN {X 0,Y 347.957,Z 541.142,A -85,B 0,C 180,E1 -13869.298,E2 -13869.298} C_VEL
LIN {X 0,Y 347.882,Z 541.153,A -85,B 0,C 180,E1 -13872.839,E2 -13872.839} C_VEL
LIN {X 0,Y 347.827,Z 541.162,A -85,B 0,C 180,E1 -13876.431,E2 -13876.431} C_VEL
LIN {X 0,Y 347.838,Z 541.159,A -85,B 0,C 180,E1 -13878.861,E2 -13878.861} C_VEL
LIN {X 0,Y 347.773,Z 541.17,A -85,B 0,C 180,E1 -13882.309,E2 -13882.309} C_VEL
LIN {X 0,Y 349.92,Z 550.893,A -85,B 0,C 180,E1 -13885.582,E2 -13885.582} C_VEL
LIN {X 0,Y 350.45,Z 553.347,A -85,B 0,C 180,E1 -13886.38,E2 -13886.38} C_VEL
LIN {X 0,Y 355.337,Z 565.528,A -85,B 0,C 180,E1 -13887.09,E2 -13887.09} C_VEL
LIN {X 0,Y 358.465,Z 580.631,A -85,B 0,C 180,E1 -13887.699,E2 -13887.699} C_VEL
LIN {X 0,Y 356.451,Z 660.55,A -85,B 0,C 180,E1 -13889.462,E2 -13889.462} C_VEL
LIN {X 0,Y 355.794,Z 673.827,A -85,B 0,C 180,E1 -13889.982,E2 -13889.982} C_VEL
LIN {X 0,Y 355.023,Z 685.671,A -85,B 0,C 180,E1 -13890.661,E2 -13890.661} C_VEL
LIN {X 0,Y 353.906,Z 697.693,A -85,B 0,C 180,E1 -13891.581,E2 -13891.581} C_VEL
LIN {X 0,Y 352.639,Z 709.974,A -85,B 0,C 180,E1 -13892.817,E2 -13892.817} C_VEL
LIN {X 0,Y 351.478,Z 719.696,A -85,B 0,C 180,E1 -13894.046,E2 -13894.046} C_VEL
LIN {X 0,Y 350.22,Z 729.475,A -85,B 0,C 180,E1 -13895.587,E2 -13895.587} C_VEL
LIN {X 0,Y 349.001,Z 738.652,A -85,B 0,C 180,E1 -13897.396,E2 -13897.396} C_VEL
LIN {X 0,Y 347.999,Z 746.118,A -85,B 0,C 180,E1 -13899.272,E2 -13899.272} C_VEL
LIN {X 0,Y 347.347,Z 751.297,A -85,B 0,C 180,E1 -13900.904,E2 -13900.904} C_VEL
LIN {X 0,Y 346.87,Z 755.423,A -85,B 0,C 180,E1 -13902.537,E2 -13902.537} C_VEL
LIN {X 0,Y 346.383,Z 759.507,A -85,B 0,C 180,E1 -13904.757,E2 -13904.757} C_VEL
LIN {X 0,Y 346.047,Z 762.043,A -85,B 0,C 180,E1 -13906.981,E2 -13906.981} C_VEL
LIN {X 0,Y 345.916,Z 762.973,A -85,B 0,C 180,E1 -13908.74,E2 -13908.74} C_VEL
LIN {X 0,Y 345.883,Z 762.809,A -85,B 0,C 180,E1 -13910.961,E2 -13910.961} C_VEL
LIN {X 0,Y 345.94,Z 761.912,A -85,B 0,C 180,E1 -13912.451,E2 -13912.451} C_VEL
LIN {X 0,Y 346.184,Z 759.839,A -85,B 0,C 180,E1 -13914.296,E2 -13914.296} C_VEL
LIN {X 0,Y 346.437,Z 756.391,A -85,B 0,C 180,E1 -13916.277,E2 -13916.277} C_VEL
LIN {X 0,Y 346.914,Z 751.441,A -85,B 0,C 180,E1 -13918.304,E2 -13918.304} C_VEL
LIN {X 0,Y 347.458,Z 745.9,A -85,B 0,C 180,E1 -13920.047,E2 -13920.047} C_VEL
LIN {X 0,Y 348.179,Z 739.407,A -85,B 0,C 180,E1 -13921.685,E2 -13921.685} C_VEL
LIN {X 0,Y 349.048,Z 731.066,A -85,B 0,C 180,E1 -13923.387,E2 -13923.387} C_VEL
LIN {X 0,Y 350.06,Z 722.028,A -85,B 0,C 180,E1 -13924.868,E2 -13924.868} C_VEL
LIN {X 0,Y 350.991,Z 713.013,A -85,B 0,C 180,E1 -13926.081,E2 -13926.081} C_VEL
LIN {X 0,Y 352.05,Z 701.862,A -85,B 0,C 180,E1 -13927.298,E2 -13927.298} C_VEL
LIN {X 0,Y 352.976,Z 689.986,A -85,B 0,C 180,E1 -13928.312,E2 -13928.312} C_VEL
LIN {X 0,Y 353.875,Z 677.063,A -85,B 0,C 180,E1 -13929.133,E2 -13929.133} C_VEL
LIN {X 0,Y 354.509,Z 664.385,A -85,B 0,C 180,E1 -13929.702,E2 -13929.702} C_VEL
LIN {X 0,Y 354.928,Z 649.213,A -85,B 0,C 180,E1 -13930.105,E2 -13930.105} C_VEL
LIN {X 0,Y 356.284,Z 579.125,A -85,B 0,C 180,E1 -13931.604,E2 -13931.604} C_VEL
LIN {X 0,Y 352.24,Z 559.02,A -85,B 0,C 180,E1 -13932.299,E2 -13932.299} C_VEL
LIN {X 0,Y 349.976,Z 552.16,A -85,B 0,C 180,E1 -13932.622,E2 -13932.622} C_VEL
LIN {X 0,Y 347.924,Z 541.145,A -85,B 0,C 180,E1 -13935.974,E2 -13935.974} C_VEL
LIN {X 0,Y 347.923,Z 541.143,A -85,B 0,C 180,E1 -13939.527,E2 -13939.527} C_VEL
LIN {X 0,Y 348.087,Z 541.126,A -85,B 0,C 180,E1 -13943.044,E2 -13943.044} C_VEL
LIN {X 0,Y 348.205,Z 541.108,A -85,B 0,C 180,E1 -13947.688,E2 -13947.688} C_VEL
LIN {X 0,Y 348.343,Z 541.09,A -85,B 0,C 180,E1 -13950.002,E2 -13950.002} C_VEL
LIN {X 0,Y 348.205,Z 541.108,A -85,B 0,C 180,E1 -13952.315,E2 -13952.315} C_VEL
LIN {X 0,Y 348.089,Z 541.128,A -85,B 0,C 180,E1 -13956.96,E2 -13956.96} C_VEL
LIN {X 0,Y 347.927,Z 541.143,A -85,B 0,C 180,E1 -13960.476,E2 -13960.476} C_VEL
LIN {X 0,Y 347.897,Z 541.146,A -85,B 0,C 180,E1 -13964.151,E2 -13964.151} C_VEL
LIN {X 0,Y 347.875,Z 541.149,A -85,B 0,C 180,E1 -13968.455,E2 -13968.455} C_VEL
LIN {X 0,Y 347.151,Z 541.245,A -85,B 0,C 180,E1 -13969.421,E2 -13969.421} C_VEL
LIN {X 0,Y 344.248,Z 541.609,A -85,B 0,C 180,E1 -13970.992,E2 -13970.992} C_VEL
LIN {X 0,Y 341.826,Z 541.909,A -85,B 0,C 180,E1 -13972.264,E2 -13972.264} C_VEL
LIN {X 0,Y 340.798,Z 542.035,A -85,B 0,C 180,E1 -13973.249,E2 -13973.249} C_VEL
LIN {X 0,Y 340.719,Z 542.041,A -85,B 0,C 180,E1 -13973.582,E2 -13973.582} C_VEL
LIN {X 0,Y 340.804,Z 542.033,A -85,B 0,C 180,E1 -13976.982,E2 -13976.982} C_VEL
LIN {X 0,Y 340.699,Z 542.047,A -85,B 0,C 180,E1 -13981.046,E2 -13981.046} C_VEL
LIN {X 0,Y 340.72,Z 542.046,A -85,B 0,C 180,E1 -13985.28,E2 -13985.28} C_VEL
LIN {X 0,Y 340.712,Z 542.041,A -85,B 0,C 180,E1 -13988.387,E2 -13988.387} C_VEL
LIN {X 0,Y 340.702,Z 542.043,A -85,B 0,C 180,E1 -13992.047,E2 -13992.047} C_VEL
LIN {X 0,Y 340.687,Z 542.049,A -85,B 0,C 180,E1 -13995.463,E2 -13995.463} C_VEL
LIN {X 0,Y 340.689,Z 542.044,A -85,B 0,C 180,E1 -13998.692,E2 -13998.692} C_VEL
LIN {X 0,Y 340.737,Z 542.041,A -85,B 0,C 180,E1 -14001.774,E2 -14001.774} C_VEL
LIN {X 0,Y 340.727,Z 542.044,A -85,B 0,C 180,E1 -14005.597,E2 -14005.597} C_VEL
LIN {X 0,Y 340.708,Z 542.042,A -85,B 0,C 180,E1 -14008.957,E2 -14008.957} C_VEL
LIN {X 0,Y 340.784,Z 542.032,A -85,B 0,C 180,E1 -14012.475,E2 -14012.475} C_VEL
LIN {X 0,Y 340.76,Z 542.041,A -85,B 0,C 180,E1 -14015.639,E2 -14015.639} C_VEL
LIN {X 0,Y 340.737,Z 542.042,A -85,B 0,C 180,E1 -14019.474,E2 -14019.474} C_VEL
LIN {X 0,Y 340.798,Z 542.033,A -85,B 0,C 180,E1 -14021.982,E2 -14021.982} C_VEL
LIN {X 0,Y 340.876,Z 542.027,A -85,B 0,C 180,E1 -14025.706,E2 -14025.706} C_VEL
LIN {X 0,Y 340.877,Z 542.022,A -85,B 0,C 180,E1 -14029.307,E2 -14029.307} C_VEL
LIN {X 0,Y 341.066,Z 541.997,A -85,B 0,C 180,E1 -14032.899,E2 -14032.899} C_VEL
LIN {X 0,Y 341.175,Z 541.988,A -85,B 0,C 180,E1 -14037.639,E2 -14037.639} C_VEL
LIN {X 0,Y 341.302,Z 541.972,A -85,B 0,C 180,E1 -14040.001,E2 -14040.001} C_VEL
LIN {X 0,Y 341.175,Z 541.985,A -85,B 0,C 180,E1 -14042.362,E2 -14042.362} C_VEL
LIN {X 0,Y 341.084,Z 541.995,A -85,B 0,C 180,E1 -14047.102,E2 -14047.102} C_VEL
LIN {X 0,Y 340.879,Z 542.02,A -85,B 0,C 180,E1 -14050.694,E2 -14050.694} C_VEL
LIN {X 0,Y 340.872,Z 542.024,A -85,B 0,C 180,E1 -14054.325,E2 -14054.325} C_VEL
LIN {X 0,Y 340.846,Z 542.026,A -85,B 0,C 180,E1 -14058.467,E2 -14058.467} C_VEL
LIN {X 0,Y 340.726,Z 542.043,A -85,B 0,C 180,E1 -14061.842,E2 -14061.842} C_VEL
LIN {X 0,Y 340.78,Z 542.034,A -85,B 0,C 180,E1 -14065.664,E2 -14065.664} C_VEL
LIN {X 0,Y 340.737,Z 542.042,A -85,B 0,C 180,E1 -14068.321,E2 -14068.321} C_VEL
LIN {X 0,Y 340.706,Z 542.042,A -85,B 0,C 180,E1 -14071.044,E2 -14071.044} C_VEL
LIN {X 0,Y 340.726,Z 542.039,A -85,B 0,C 180,E1 -14075.279,E2 -14075.279} C_VEL
LIN {X 0,Y 340.717,Z 542.045,A -85,B 0,C 180,E1 -14078.385,E2 -14078.385} C_VEL
LIN {X 0,Y 340.706,Z 542.046,A -85,B 0,C 180,E1 -14082.045,E2 -14082.045} C_VEL
LIN {X 0,Y 340.66,Z 542.053,A -85,B 0,C 180,E1 -14086.226,E2 -14086.226} C_VEL
LIN {X 0,Y 340.696,Z 542.044,A -85,B 0,C 180,E1 -14089.752,E2 -14089.752} C_VEL
LIN {X 0,Y 340.715,Z 542.04,A -85,B 0,C 180,E1 -14093.258,E2 -14093.258} C_VEL
LIN {X 0,Y 340.7,Z 542.046,A -85,B 0,C 180,E1 -14096.153,E2 -14096.153} C_VEL
LIN {X 0,Y 340.756,Z 542.083,A -85,B 0,C 180,E1 -14099.371,E2 -14099.371} C_VEL
LIN {X 0,Y 343.155,Z 553.438,A -85,B 0,C 180,E1 -14102.559,E2 -14102.559} C_VEL
LIN {X 0,Y 344.615,Z 561.127,A -85,B 0,C 180,E1 -14104.641,E2 -14104.641} C_VEL
LIN {X 0,Y 344.512,Z 564.917,A -85,B 0,C 180,E1 -14105.599,E2 -14105.599} C_VEL
LIN {X 0,Y 343.885,Z 570.786,A -85,B 0,C 180,E1 -14107.046,E2 -14107.046} C_VEL
LIN {X 0,Y 349.344,Z 606.663,A -85,B 0,C 180,E1 -14108.218,E2 -14108.218} C_VEL
LIN {X 0,Y 347.802,Z 679.333,A -85,B 0,C 180,E1 -14109.83,E2 -14109.83} C_VEL
LIN {X 0,Y 347.03,Z 692.961,A -85,B 0,C 180,E1 -14110.362,E2 -14110.362} C_VEL
LIN {X 0,Y 346.199,Z 704.813,A -85,B 0,C 180,E1 -14111.045,E2 -14111.045} C_VEL
LIN {X 0,Y 345.222,Z 716.094,A -85,B 0,C 180,E1 -14111.912,E2 -14111.912} C_VEL
LIN {X 0,Y 344.047,Z 727.782,A -85,B 0,C 180,E1 -14113.075,E2 -14113.075} C_VEL
LIN {X 0,Y 342.877,Z 738.692,A -85,B 0,C 180,E1 -14114.445,E2 -14114.445} C_VEL
LIN {X 0,Y 342.018,Z 746.933,A -85,B 0,C 180,E1 -14115.723,E2 -14115.723} C_VEL
LIN {X 0,Y 341.121,Z 754.868,A -85,B 0,C 180,E1 -14117.203,E2 -14117.203} C_VEL
LIN {X 0,Y 340.284,Z 762.598,A -85,B 0,C 180,E1 -14118.985,E2 -14118.985} C_VEL
LIN {X 0,Y 339.786,Z 767.885,A -85,B 0,C 180,E1 -14120.474,E2 -14120.474} C_VEL
LIN {X 0,Y 339.4,Z 772.99,A -85,B 0,C 180,E1 -14122.263,E2 -14122.263} C_VEL
LIN {X 0,Y 339.154,Z 776.988,A -85,B 0,C 180,E1 -14124.083,E2 -14124.083} C_VEL
LIN {X 0,Y 339.099,Z 778.951,A -85,B 0,C 180,E1 -14125.243,E2 -14125.243} C_VEL
LIN {X 0,Y 339.075,Z 780.548,A -85,B 0,C 180,E1 -14126.433,E2 -14126.433} C_VEL
LIN {X 0,Y 339.002,Z 781.713,A -85,B 0,C 180,E1 -14127.622,E2 -14127.622} C_VEL
LIN {X 0,Y 339.021,Z 782.431,A -85,B 0,C 180,E1 -14128.81,E2 -14128.81} C_VEL
LIN {X 0,Y 339.068,Z 782.753,A -85,B 0,C 180,E1 -14129.998,E2 -14129.998} C_VEL
LIN {X 0,Y 339.007,Z 782.676,A -85,B 0,C 180,E1 -14131.186,E2 -14131.186} C_VEL
LIN {X 0,Y 338.999,Z 782.19,A -85,B 0,C 180,E1 -14132.375,E2 -14132.375} C_VEL
LIN {X 0,Y 339.072,Z 781.266,A -85,B 0,C 180,E1 -14133.563,E2 -14133.563} C_VEL
LIN {X 0,Y 339.113,Z 778.349,A -85,B 0,C 180,E1 -14135.85,E2 -14135.85} C_VEL
LIN {X 0,Y 339.401,Z 774.719,A -85,B 0,C 180,E1 -14137.733,E2 -14137.733} C_VEL
LIN {X 0,Y 339.835,Z 770.157,A -85,B 0,C 180,E1 -14139.521,E2 -14139.521} C_VEL
LIN {X 0,Y 340.513,Z 764.383,A -85,B 0,C 180,E1 -14141.306,E2 -14141.306} C_VEL
LIN {X 0,Y 341.493,Z 757.155,A -85,B 0,C 180,E1 -14143.082,E2 -14143.082} C_VEL
LIN {X 0,Y 342.757,Z 748.182,A -85,B 0,C 180,E1 -14144.849,E2 -14144.849} C_VEL
LIN {X 0,Y 344.011,Z 738.096,A -85,B 0,C 180,E1 -14146.447,E2 -14146.447} C_VEL
LIN {X 0,Y 345.334,Z 727.553,A -85,B 0,C 180,E1 -14147.772,E2 -14147.772} C_VEL
LIN {X 0,Y 346.692,Z 716.035,A -85,B 0,C 180,E1 -14148.924,E2 -14148.924} C_VEL
LIN {X 0,Y 347.898,Z 703.983,A -85,B 0,C 180,E1 -14149.853,E2 -14149.853} C_VEL
LIN {X 0,Y 348.939,Z 691.466,A -85,B 0,C 180,E1 -14150.559,E2 -14150.559} C_VEL
LIN {X 0,Y 349.682,Z 678.751,A -85,B 0,C 180,E1 -14151.053,E2 -14151.053} C_VEL
LIN {X 0,Y 351.476,Z 606.382,A -85,B 0,C 180,E1 -14152.693,E2 -14152.693} C_VEL
LIN {X 0,Y 348.075,Z 584.808,A -85,B 0,C 180,E1 -14153.498,E2 -14153.498} C_VEL
LIN {X 0,Y 344.972,Z 569.756,A -85,B 0,C 180,E1 -14154.143,E2 -14154.143} C_VEL
LIN {X 0,Y 345.5,Z 565.277,A -85,B 0,C 180,E1 -14155.286,E2 -14155.286} C_VEL
LIN {X 0,Y 344.369,Z 558.076,A -85,B 0,C 180,E1 -14157.333,E2 -14157.333} C_VEL
LIN {X 0,Y 342.197,Z 547.959,A -85,B 0,C 180,E1 -14160.39,E2 -14160.39} C_VEL
LIN {X 0,Y 340.678,Z 542.048,A -85,B 0,C 180,E1 -14162.322,E2 -14162.322} C_VEL
LIN {X 0,Y 340.715,Z 542.046,A -85,B 0,C 180,E1 -14165.277,E2 -14165.277} C_VEL
LIN {X 0,Y 340.715,Z 542.047,A -85,B 0,C 180,E1 -14168.386,E2 -14168.386} C_VEL
LIN {X 0,Y 340.726,Z 542.047,A -85,B 0,C 180,E1 -14172.05,E2 -14172.05} C_VEL
LIN {X 0,Y 340.668,Z 542.052,A -85,B 0,C 180,E1 -14176.221,E2 -14176.221} C_VEL
LIN {X 0,Y 340.698,Z 542.047,A -85,B 0,C 180,E1 -14178.692,E2 -14178.692} C_VEL
LIN {X 0,Y 340.732,Z 542.04,A -85,B 0,C 180,E1 -14181.772,E2 -14181.772} C_VEL
LIN {X 0,Y 340.715,Z 542.04,A -85,B 0,C 180,E1 -14185.594,E2 -14185.594} C_VEL
LIN {X 0,Y 340.696,Z 542.042,A -85,B 0,C 180,E1 -14188.954,E2 -14188.954} C_VEL
LIN {X 0,Y 340.771,Z 542.031,A -85,B 0,C 180,E1 -14192.472,E2 -14192.472} C_VEL
LIN {X 0,Y 340.746,Z 542.036,A -85,B 0,C 180,E1 -14195.637,E2 -14195.637} C_VEL
LIN {X 0,Y 340.738,Z 542.037,A -85,B 0,C 180,E1 -14199.473,E2 -14199.473} C_VEL
LIN {X 0,Y 340.848,Z 542.027,A -85,B 0,C 180,E1 -14201.983,E2 -14201.983} C_VEL
LIN {X 0,Y 340.858,Z 542.028,A -85,B 0,C 180,E1 -14205.704,E2 -14205.704} C_VEL
LIN {X 0,Y 340.864,Z 542.023,A -85,B 0,C 180,E1 -14209.305,E2 -14209.305} C_VEL
LIN {X 0,Y 341.064,Z 541.997,A -85,B 0,C 180,E1 -14212.897,E2 -14212.897} C_VEL
LIN {X 0,Y 341.16,Z 541.988,A -85,B 0,C 180,E1 -14217.638,E2 -14217.638} C_VEL
LIN {X 0,Y 341.306,Z 541.971,A -85,B 0,C 180,E1 -14219.999,E2 -14219.999} C_VEL
LIN {X 0,Y 341.16,Z 541.986,A -85,B 0,C 180,E1 -14222.361,E2 -14222.361} C_VEL
LIN {X 0,Y 341.067,Z 541.999,A -85,B 0,C 180,E1 -14227.101,E2 -14227.101} C_VEL
LIN {X 0,Y 340.864,Z 542.025,A -85,B 0,C 180,E1 -14230.693,E2 -14230.693} C_VEL
LIN {X 0,Y 340.85,Z 542.03,A -85,B 0,C 180,E1 -14234.325,E2 -14234.325} C_VEL
LIN {X 0,Y 340.824,Z 542.032,A -85,B 0,C 180,E1 -14238.466,E2 -14238.466} C_VEL
LIN {X 0,Y 340.732,Z 542.072,A -85,B 0,C 180,E1 -14241.793,E2 -14241.793} C_VEL
LIN {X 0,Y 342.715,Z 550.905,A -85,B 0,C 180,E1 -14244.859,E2 -14244.859} C_VEL
LIN {X 0,Y 343.328,Z 553.745,A -85,B 0,C 180,E1 -14245.784,E2 -14245.784} C_VEL
LIN {X 0,Y 349.33,Z 568.417,A -85,B 0,C 180,E1 -14246.672,E2 -14246.672} C_VEL
LIN {X 0,Y 352.026,Z 581.432,A -85,B 0,C 180,E1 -14247.213,E2 -14247.213} C_VEL
LIN {X 0,Y 349.937,Z 660.829,A -85,B 0,C 180,E1 -14249.011,E2 -14249.011} C_VEL
LIN {X 0,Y 349.252,Z 674.011,A -85,B 0,C 180,E1 -14249.538,E2 -14249.538} C_VEL
LIN {X 0,Y 348.361,Z 686.772,A -85,B 0,C 180,E1 -14250.288,E2 -14250.288} C_VEL
LIN {X 0,Y 347.202,Z 698.747,A -85,B 0,C 180,E1 -14251.244,E2 -14251.244} C_VEL
LIN {X 0,Y 345.996,Z 709.915,A -85,B 0,C 180,E1 -14252.393,E2 -14252.393} C_VEL
LIN {X 0,Y 344.664,Z 720.462,A -85,B 0,C 180,E1 -14253.754,E2 -14253.754} C_VEL
LIN {X 0,Y 343.329,Z 730.346,A -85,B 0,C 180,E1 -14255.363,E2 -14255.363} C_VEL
LIN {X 0,Y 342.136,Z 738.73,A -85,B 0,C 180,E1 -14257.056,E2 -14257.056} C_VEL
LIN {X 0,Y 341.176,Z 745.486,A -85,B 0,C 180,E1 -14258.751,E2 -14258.751} C_VEL
LIN {X 0,Y 340.318,Z 751.754,A -85,B 0,C 180,E1 -14260.756,E2 -14260.756} C_VEL
LIN {X 0,Y 339.816,Z 755.853,A -85,B 0,C 180,E1 -14262.439,E2 -14262.439} C_VEL
LIN {X 0,Y 339.541,Z 758.074,A -85,B 0,C 180,E1 -14263.58,E2 -14263.58} C_VEL
LIN {X 0,Y 339.207,Z 760.553,A -85,B 0,C 180,E1 -14265.218,E2 -14265.218} C_VEL
LIN {X 0,Y 338.986,Z 762.223,A -85,B 0,C 180,E1 -14266.832,E2 -14266.832} C_VEL
LIN {X 0,Y 338.84,Z 763.088,A -85,B 0,C 180,E1 -14268.418,E2 -14268.418} C_VEL
LIN {X 0,Y 338.754,Z 763.231,A -85,B 0,C 180,E1 -14270.14,E2 -14270.14} C_VEL
LIN {X 0,Y 338.815,Z 762.424,A -85,B 0,C 180,E1 -14272.019,E2 -14272.019} C_VEL
LIN {X 0,Y 339.03,Z 760.537,A -85,B 0,C 180,E1 -14273.944,E2 -14273.944} C_VEL
LIN {X 0,Y 339.306,Z 757.299,A -85,B 0,C 180,E1 -14275.999,E2 -14275.999} C_VEL
LIN {X 0,Y 339.735,Z 752.785,A -85,B 0,C 180,E1 -14278.01,E2 -14278.01} C_VEL
LIN {X 0,Y 340.213,Z 748.286,A -85,B 0,C 180,E1 -14279.556,E2 -14279.556} C_VEL
LIN {X 0,Y 340.943,Z 741.748,A -85,B 0,C 180,E1 -14281.365,E2 -14281.365} C_VEL
LIN {X 0,Y 341.796,Z 733.857,A -85,B 0,C 180,E1 -14283.107,E2 -14283.107} C_VEL
LIN {X 0,Y 342.806,Z 725.148,A -85,B 0,C 180,E1 -14284.663,E2 -14284.663} C_VEL
LIN {X 0,Y 343.831,Z 715.388,A -85,B 0,C 180,E1 -14286.086,E2 -14286.086} C_VEL
LIN {X 0,Y 344.839,Z 705.758,A -85,B 0,C 180,E1 -14287.22,E2 -14287.22} C_VEL
LIN {X 0,Y 345.772,Z 695.161,A -85,B 0,C 180,E1 -14288.228,E2 -14288.228} C_VEL
LIN {X 0,Y 346.735,Z 682.71,A -85,B 0,C 180,E1 -14289.144,E2 -14289.144} C_VEL
LIN {X 0,Y 347.482,Z 669.394,A -85,B 0,C 180,E1 -14289.855,E2 -14289.855} C_VEL
LIN {X 0,Y 347.994,Z 655.997,A -85,B 0,C 180,E1 -14290.307,E2 -14290.307} C_VEL
LIN {X 0,Y 349.583,Z 579.935,A -85,B 0,C 180,E1 -14291.972,E2 -14291.972} C_VEL
LIN {X 0,Y 345.744,Z 561.088,A -85,B 0,C 180,E1 -14292.642,E2 -14292.642} C_VEL
LIN {X 0,Y 342.833,Z 552.407,A -85,B 0,C 180,E1 -14293.048,E2 -14293.048} C_VEL
LIN {X 0,Y 340.879,Z 542.023,A -85,B 0,C 180,E1 -14296.286,E2 -14296.286} C_VEL
LIN {X 0,Y 340.921,Z 542.018,A -85,B 0,C 180,E1 -14300.509,E2 -14300.509} C_VEL
LIN {X 0,Y 341.055,Z 542.004,A -85,B 0,C 180,E1 -14302.9,E2 -14302.9} C_VEL
LIN {X 0,Y 341.167,Z 541.984,A -85,B 0,C 180,E1 -14307.64,E2 -14307.64} C_VEL
LIN {X 0,Y 341.294,Z 541.968,A -85,B 0,C 180,E1 -14310.002,E2 -14310.002} C_VEL
LIN {X 0,Y 341.167,Z 541.985,A -85,B 0,C 180,E1 -14312.363,E2 -14312.363} C_VEL
LIN {X 0,Y 341.058,Z 542.003,A -85,B 0,C 180,E1 -14317.104,E2 -14317.104} C_VEL
LIN {X 0,Y 340.87,Z 542.024,A -85,B 0,C 180,E1 -14320.695,E2 -14320.695} C_VEL
LIN {X 0,Y 340.862,Z 542.022,A -85,B 0,C 180,E1 -14324.326,E2 -14324.326} C_VEL
LIN {X 0,Y 340.836,Z 542.026,A -85,B 0,C 180,E1 -14328.468,E2 -14328.468} C_VEL
LIN {X 0,Y 340.754,Z 542.036,A -85,B 0,C 180,E1 -14331.859,E2 -14331.859} C_VEL
LIN {X 0,Y 340.719,Z 542.041,A -85,B 0,C 180,E1 -14333.582,E2 -14333.582} C_VEL
LIN {X 0,Y 340.06,Z 542.124,A -85,B 0,C 180,E1 -14334.569,E2 -14334.569} C_VEL
LIN {X 0,Y 337.203,Z 542.478,A -85,B 0,C 180,E1 -14336.174,E2 -14336.174} C_VEL
LIN {X 0,Y 334.785,Z 542.783,A -85,B 0,C 180,E1 -14337.473,E2 -14337.473} C_VEL
LIN {X 0,Y 333.762,Z 542.908,A -85,B 0,C 180,E1 -14338.479,E2 -14338.479} C_VEL
LIN {X 0,Y 333.686,Z 542.918,A -85,B 0,C 180,E1 -14338.82,E2 -14338.82} C_VEL
LIN {X 0,Y 333.645,Z 542.922,A -85,B 0,C 180,E1 -14342.589,E2 -14342.589} C_VEL
LIN {X 0,Y 333.678,Z 542.917,A -85,B 0,C 180,E1 -14346.141,E2 -14346.141} C_VEL
LIN {X 0,Y 333.649,Z 542.926,A -85,B 0,C 180,E1 -14349.194,E2 -14349.194} C_VEL
LIN {X 0,Y 333.635,Z 542.922,A -85,B 0,C 180,E1 -14352.502,E2 -14352.502} C_VEL
LIN {X 0,Y 333.625,Z 542.925,A -85,B 0,C 180,E1 -14355.961,E2 -14355.961} C_VEL
LIN {X 0,Y 333.651,Z 542.926,A -85,B 0,C 180,E1 -14359.317,E2 -14359.317} C_VEL
LIN {X 0,Y 333.669,Z 542.921,A -85,B 0,C 180,E1 -14363.169,E2 -14363.169} C_VEL
LIN {X 0,Y 333.678,Z 542.922,A -85,B 0,C 180,E1 -14365.343,E2 -14365.343} C_VEL
LIN {X 0,Y 333.708,Z 542.917,A -85,B 0,C 180,E1 -14369.712,E2 -14369.712} C_VEL
LIN {X 0,Y 333.749,Z 542.908,A -85,B 0,C 180,E1 -14372.402,E2 -14372.402} C_VEL
LIN {X 0,Y 333.731,Z 542.912,A -85,B 0,C 180,E1 -14375.092,E2 -14375.092} C_VEL
LIN {X 0,Y 333.677,Z 542.918,A -85,B 0,C 180,E1 -14379.02,E2 -14379.02} C_VEL
LIN {X 0,Y 333.747,Z 542.914,A -85,B 0,C 180,E1 -14381.587,E2 -14381.587} C_VEL
LIN {X 0,Y 333.815,Z 542.905,A -85,B 0,C 180,E1 -14385.578,E2 -14385.578} C_VEL
LIN {X 0,Y 333.84,Z 542.898,A -85,B 0,C 180,E1 -14389.079,E2 -14389.079} C_VEL
LIN {X 0,Y 334.013,Z 542.875,A -85,B 0,C 180,E1 -14392.748,E2 -14392.748} C_VEL
LIN {X 0,Y 333.815,Z 542.901,A -85,B 0,C 180,E1 -14395.17,E2 -14395.17} C_VEL
LIN {X 0,Y 334.112,Z 542.867,A -85,B 0,C 180,E1 -14397.589,E2 -14397.589} C_VEL
LIN {X 0,Y 334.253,Z 542.85,A -85,B 0,C 180,E1 -14400.001,E2 -14400.001} C_VEL
LIN {X 0,Y 334.112,Z 542.864,A -85,B 0,C 180,E1 -14402.412,E2 -14402.412} C_VEL
LIN {X 0,Y 334.034,Z 542.873,A -85,B 0,C 180,E1 -14407.253,E2 -14407.253} C_VEL
LIN {X 0,Y 333.842,Z 542.897,A -85,B 0,C 180,E1 -14410.922,E2 -14410.922} C_VEL
LIN {X 0,Y 333.817,Z 542.9,A -85,B 0,C 180,E1 -14414.634,E2 -14414.634} C_VEL
LIN {X 0,Y 333.805,Z 542.902,A -85,B 0,C 180,E1 -14418.655,E2 -14418.655} C_VEL
LIN {X 0,Y 333.665,Z 542.922,A -85,B 0,C 180,E1 -14422.281,E2 -14422.281} C_VEL
LIN {X 0,Y 333.743,Z 542.913,A -85,B 0,C 180,E1 -14426.246,E2 -14426.246} C_VEL
LIN {X 0,Y 333.698,Z 542.915,A -85,B 0,C 180,E1 -14428.974,E2 -14428.974} C_VEL
LIN {X 0,Y 333.652,Z 542.922,A -85,B 0,C 180,E1 -14432.587,E2 -14432.587} C_VEL
LIN {X 0,Y 333.684,Z 542.922,A -85,B 0,C 180,E1 -14436.139,E2 -14436.139} C_VEL
LIN {X 0,Y 333.655,Z 542.92,A -85,B 0,C 180,E1 -14439.192,E2 -14439.192} C_VEL
LIN {X 0,Y 333.64,Z 542.925,A -85,B 0,C 180,E1 -14442.499,E2 -14442.499} C_VEL
LIN {X 0,Y 333.604,Z 542.929,A -85,B 0,C 180,E1 -14445.954,E2 -14445.954} C_VEL
LIN {X 0,Y 333.655,Z 542.92,A -85,B 0,C 180,E1 -14449.315,E2 -14449.315} C_VEL
LIN {X 0,Y 333.675,Z 542.918,A -85,B 0,C 180,E1 -14453.167,E2 -14453.167} C_VEL
LIN {X 0,Y 333.644,Z 542.924,A -85,B 0,C 180,E1 -14456.791,E2 -14456.791} C_VEL
LIN {X 0,Y 333.712,Z 542.984,A -85,B 0,C 180,E1 -14459.033,E2 -14459.033} C_VEL
LIN {X 0,Y 336.004,Z 553.666,A -85,B 0,C 180,E1 -14462.111,E2 -14462.111} C_VEL
LIN {X 0,Y 337.577,Z 561.951,A -85,B 0,C 180,E1 -14464.404,E2 -14464.404} C_VEL
LIN {X 0,Y 337.573,Z 565.75,A -85,B 0,C 180,E1 -14465.392,E2 -14465.392} C_VEL
LIN {X 0,Y 337.024,Z 570.635,A -85,B 0,C 180,E1 -14466.621,E2 -14466.621} C_VEL
LIN {X 0,Y 342.631,Z 606.972,A -85,B 0,C 180,E1 -14467.836,E2 -14467.836} C_VEL
LIN {X 0,Y 341.021,Z 679.698,A -85,B 0,C 180,E1 -14469.49,E2 -14469.49} C_VEL
LIN {X 0,Y 340.225,Z 693.132,A -85,B 0,C 180,E1 -14470.031,E2 -14470.031} C_VEL
LIN {X 0,Y 339.268,Z 705.929,A -85,B 0,C 180,E1 -14470.799,E2 -14470.799} C_VEL
LIN {X 0,Y 338.101,Z 718.472,A -85,B 0,C 180,E1 -14471.831,E2 -14471.831} C_VEL
LIN {X 0,Y 336.9,Z 729.696,A -85,B 0,C 180,E1 -14473.018,E2 -14473.018} C_VEL
LIN {X 0,Y 335.902,Z 739.028,A -85,B 0,C 180,E1 -14474.25,E2 -14474.25} C_VEL
LIN {X 0,Y 334.883,Z 748.12,A -85,B 0,C 180,E1 -14475.722,E2 -14475.722} C_VEL
LIN {X 0,Y 333.985,Z 755.802,A -85,B 0,C 180,E1 -14477.234,E2 -14477.234} C_VEL
LIN {X 0,Y 333.155,Z 763.328,A -85,B 0,C 180,E1 -14479.054,E2 -14479.054} C_VEL
LIN {X 0,Y 332.579,Z 769.359,A -85,B 0,C 180,E1 -14480.879,E2 -14480.879} C_VEL
LIN {X 0,Y 332.243,Z 774.109,A -85,B 0,C 180,E1 -14482.707,E2 -14482.707} C_VEL
LIN {X 0,Y 332.047,Z 777.038,A -85,B 0,C 180,E1 -14484.152,E2 -14484.152} C_VEL
LIN {X 0,Y 332.002,Z 780.283,A -85,B 0,C 180,E1 -14486.357,E2 -14486.357} C_VEL
LIN {X 0,Y 331.919,Z 781.471,A -85,B 0,C 180,E1 -14487.571,E2 -14487.571} C_VEL
LIN {X 0,Y 331.926,Z 782.206,A -85,B 0,C 180,E1 -14488.785,E2 -14488.785} C_VEL
LIN {X 0,Y 331.971,Z 782.54,A -85,B 0,C 180,E1 -14489.998,E2 -14489.998} C_VEL
LIN {X 0,Y 331.913,Z 782.476,A -85,B 0,C 180,E1 -14491.212,E2 -14491.212} C_VEL
LIN {X 0,Y 331.917,Z 782.012,A -85,B 0,C 180,E1 -14492.425,E2 -14492.425} C_VEL
LIN {X 0,Y 331.975,Z 781.103,A -85,B 0,C 180,E1 -14493.64,E2 -14493.64} C_VEL
LIN {X 0,Y 332.01,Z 778.505,A -85,B 0,C 180,E1 -14495.785,E2 -14495.785} C_VEL
LIN {X 0,Y 332.358,Z 774.621,A -85,B 0,C 180,E1 -14497.898,E2 -14497.898} C_VEL
LIN {X 0,Y 332.809,Z 770.089,A -85,B 0,C 180,E1 -14499.724,E2 -14499.724} C_VEL
LIN {X 0,Y 333.513,Z 764.352,A -85,B 0,C 180,E1 -14501.546,E2 -14501.546} C_VEL
LIN {X 0,Y 334.569,Z 757.176,A -85,B 0,C 180,E1 -14503.358,E2 -14503.358} C_VEL
LIN {X 0,Y 335.863,Z 748.244,A -85,B 0,C 180,E1 -14505.161,E2 -14505.161} C_VEL
LIN {X 0,Y 337.181,Z 738.405,A -85,B 0,C 180,E1 -14506.764,E2 -14506.764} C_VEL
LIN {X 0,Y 338.587,Z 727.772,A -85,B 0,C 180,E1 -14508.139,E2 -14508.139} C_VEL
LIN {X 0,Y 340.009,Z 716.381,A -85,B 0,C 180,E1 -14509.311,E2 -14509.311} C_VEL
LIN {X 0,Y 341.26,Z 704.585,A -85,B 0,C 180,E1 -14510.256,E2 -14510.256} C_VEL
LIN {X 0,Y 342.403,Z 691.67,A -85,B 0,C 180,E1 -14511.009,E2 -14511.009} C_VEL
LIN {X 0,Y 343.172,Z 679.216,A -85,B 0,C 180,E1 -14511.511,E2 -14511.511} C_VEL
LIN {X 0,Y 344.196,Z 645.335,A -85,B 0,C 180,E1 -14512.306,E2 -14512.306} C_VEL
LIN {X 0,Y 345.03,Z 606.921,A -85,B 0,C 180,E1 -14513.195,E2 -14513.195} C_VEL
LIN {X 0,Y 341.803,Z 586.425,A -85,B 0,C 180,E1 -14513.983,E2 -14513.983} C_VEL
LIN {X 0,Y 338.321,Z 569.436,A -85,B 0,C 180,E1 -14514.761,E2 -14514.761} C_VEL
LIN {X 0,Y 338.545,Z 565.411,A -85,B 0,C 180,E1 -14515.843,E2 -14515.843} C_VEL
LIN {X 0,Y 336.505,Z 554.682,A -85,B 0,C 180,E1 -14519.048,E2 -14519.048} C_VEL
LIN {X 0,Y 334.168,Z 545.079,A -85,B 0,C 180,E1 -14522.147,E2 -14522.147} C_VEL
LIN {X 0,Y 333.642,Z 542.923,A -85,B 0,C 180,E1 -14522.931,E2 -14522.931} C_VEL
LIN {X 0,Y 333.674,Z 542.924,A -85,B 0,C 180,E1 -14526.137,E2 -14526.137} C_VEL
LIN {X 0,Y 333.668,Z 542.927,A -85,B 0,C 180,E1 -14529.187,E2 -14529.187} C_VEL
LIN {X 0,Y 333.661,Z 542.925,A -85,B 0,C 180,E1 -14532.505,E2 -14532.505} C_VEL
LIN {X 0,Y 333.614,Z 542.932,A -85,B 0,C 180,E1 -14535.957,E2 -14535.957} C_VEL
LIN {X 0,Y 333.649,Z 542.923,A -85,B 0,C 180,E1 -14539.312,E2 -14539.312} C_VEL
LIN {X 0,Y 333.649,Z 542.919,A -85,B 0,C 180,E1 -14542.348,E2 -14542.348} C_VEL
LIN {X 0,Y 333.666,Z 542.919,A -85,B 0,C 180,E1 -14545.34,E2 -14545.34} C_VEL
LIN {X 0,Y 333.694,Z 542.914,A -85,B 0,C 180,E1 -14549.709,E2 -14549.709} C_VEL
LIN {X 0,Y 333.735,Z 542.907,A -85,B 0,C 180,E1 -14552.4,E2 -14552.4} C_VEL
LIN {X 0,Y 333.718,Z 542.917,A -85,B 0,C 180,E1 -14555.089,E2 -14555.089} C_VEL
LIN {X 0,Y 333.673,Z 542.922,A -85,B 0,C 180,E1 -14559.018,E2 -14559.018} C_VEL
LIN {X 0,Y 333.784,Z 542.905,A -85,B 0,C 180,E1 -14561.588,E2 -14561.588} C_VEL
LIN {X 0,Y 333.797,Z 542.905,A -85,B 0,C 180,E1 -14565.576,E2 -14565.576} C_VEL
LIN {X 0,Y 333.827,Z 542.897,A -85,B 0,C 180,E1 -14569.077,E2 -14569.077} C_VEL
LIN {X 0,Y 334.014,Z 542.874,A -85,B 0,C 180,E1 -14572.747,E2 -14572.747} C_VEL
LIN {X 0,Y 333.803,Z 542.9,A -85,B 0,C 180,E1 -14575.168,E2 -14575.168} C_VEL
LIN {X 0,Y 334.121,Z 542.865,A -85,B 0,C 180,E1 -14577.588,E2 -14577.588} C_VEL
LIN {X 0,Y 334.256,Z 542.849,A -85,B 0,C 180,E1 -14579.999,E2 -14579.999} C_VEL
LIN {X 0,Y 334.121,Z 542.862,A -85,B 0,C 180,E1 -14582.41,E2 -14582.41} C_VEL
LIN {X 0,Y 334.016,Z 542.877,A -85,B 0,C 180,E1 -14587.252,E2 -14587.252} C_VEL
LIN {X 0,Y 333.826,Z 542.903,A -85,B 0,C 180,E1 -14590.922,E2 -14590.922} C_VEL
LIN {X 0,Y 333.796,Z 542.909,A -85,B 0,C 180,E1 -14594.634,E2 -14594.634} C_VEL
LIN {X 0,Y 333.777,Z 542.91,A -85,B 0,C 180,E1 -14598.652,E2 -14598.652} C_VEL
LIN {X 0,Y 333.704,Z 542.92,A -85,B 0,C 180,E1 -14601.221,E2 -14601.221} C_VEL
LIN {X 0,Y 335.89,Z 552.774,A -85,B 0,C 180,E1 -14604.737,E2 -14604.737} C_VEL
LIN {X 0,Y 336.149,Z 553.94,A -85,B 0,C 180,E1 -14605.13,E2 -14605.13} C_VEL
LIN {X 0,Y 343.172,Z 570.452,A -85,B 0,C 180,E1 -14606.202,E2 -14606.202} C_VEL
LIN {X 0,Y 345.674,Z 583.03,A -85,B 0,C 180,E1 -14606.732,E2 -14606.732} C_VEL
LIN {X 0,Y 343.445,Z 661.475,A -85,B 0,C 180,E1 -14608.545,E2 -14608.545} C_VEL
LIN {X 0,Y 342.696,Z 674.924,A -85,B 0,C 180,E1 -14609.1,E2 -14609.1} C_VEL
LIN {X 0,Y 341.836,Z 686.513,A -85,B 0,C 180,E1 -14609.798,E2 -14609.798} C_VEL
LIN {X 0,Y 340.731,Z 697.788,A -85,B 0,C 180,E1 -14610.696,E2 -14610.696} C_VEL
LIN {X 0,Y 339.388,Z 709.452,A -85,B 0,C 180,E1 -14611.899,E2 -14611.899} C_VEL
LIN {X 0,Y 338.16,Z 719.13,A -85,B 0,C 180,E1 -14613.148,E2 -14613.148} C_VEL
LIN {X 0,Y 336.89,Z 727.969,A -85,B 0,C 180,E1 -14614.537,E2 -14614.537} C_VEL
LIN {X 0,Y 335.629,Z 736.495,A -85,B 0,C 180,E1 -14616.186,E2 -14616.186} C_VEL
LIN {X 0,Y 334.39,Z 744.712,A -85,B 0,C 180,E1 -14618.189,E2 -14618.189} C_VEL
LIN {X 0,Y 333.427,Z 751.3,A -85,B 0,C 180,E1 -14620.252,E2 -14620.252} C_VEL
LIN {X 0,Y 332.702,Z 756.69,A -85,B 0,C 180,E1 -14622.528,E2 -14622.528} C_VEL
LIN {X 0,Y 332.299,Z 759.682,A -85,B 0,C 180,E1 -14624.261,E2 -14624.261} C_VEL
LIN {X 0,Y 331.965,Z 761.835,A -85,B 0,C 180,E1 -14626.038,E2 -14626.038} C_VEL
LIN {X 0,Y 331.782,Z 763.115,A -85,B 0,C 180,E1 -14627.849,E2 -14627.849} C_VEL
LIN {X 0,Y 331.687,Z 763.496,A -85,B 0,C 180,E1 -14629.71,E2 -14629.71} C_VEL
LIN {X 0,Y 331.739,Z 762.57,A -85,B 0,C 180,E1 -14632.096,E2 -14632.096} C_VEL
LIN {X 0,Y 332.007,Z 760.211,A -85,B 0,C 180,E1 -14634.402,E2 -14634.402} C_VEL
LIN {X 0,Y 332.348,Z 756.362,A -85,B 0,C 180,E1 -14636.648,E2 -14636.648} C_VEL
LIN {X 0,Y 332.922,Z 751.011,A -85,B 0,C 180,E1 -14638.858,E2 -14638.858} C_VEL
LIN {X 0,Y 333.554,Z 745.022,A -85,B 0,C 180,E1 -14640.735,E2 -14640.735} C_VEL
LIN {X 0,Y 334.361,Z 738.12,A -85,B 0,C 180,E1 -14642.459,E2 -14642.459} C_VEL
LIN {X 0,Y 335.418,Z 729.019,A -85,B 0,C 180,E1 -14644.285,E2 -14644.285} C_VEL
LIN {X 0,Y 336.487,Z 719.74,A -85,B 0,C 180,E1 -14645.785,E2 -14645.785} C_VEL
LIN {X 0,Y 337.717,Z 708.774,A -85,B 0,C 180,E1 -14647.197,E2 -14647.197} C_VEL
LIN {X 0,Y 338.813,Z 697.267,A -85,B 0,C 180,E1 -14648.376,E2 -14648.376} C_VEL
LIN {X 0,Y 339.764,Z 685.495,A -85,B 0,C 180,E1 -14649.309,E2 -14649.309} C_VEL
LIN {X 0,Y 340.574,Z 671.911,A -85,B 0,C 180,E1 -14650.095,E2 -14650.095} C_VEL
LIN {X 0,Y 341.179,Z 658.613,A -85,B 0,C 180,E1 -14650.602,E2 -14650.602} C_VEL
LIN {X 0,Y 342.99,Z 581.348,A -85,B 0,C 180,E1 -14652.333,E2 -14652.333} C_VEL
LIN {X 0,Y 339.231,Z 562.951,A -85,B 0,C 180,E1 -14653.006,E2 -14653.006} C_VEL
LIN {X 0,Y 335.632,Z 552.572,A -85,B 0,C 180,E1 -14653.515,E2 -14653.515} C_VEL
LIN {X 0,Y 333.816,Z 542.905,A -85,B 0,C 180,E1 -14656.611,E2 -14656.611} C_VEL
LIN {X 0,Y 333.856,Z 542.896,A -85,B 0,C 180,E1 -14660.307,E2 -14660.307} C_VEL
LIN {X 0,Y 334.008,Z 542.881,A -85,B 0,C 180,E1 -14662.749,E2 -14662.749} C_VEL
LIN {X 0,Y 333.807,Z 542.904,A -85,B 0,C 180,E1 -14665.171,E2 -14665.171} C_VEL
LIN {X 0,Y 334.104,Z 542.865,A -85,B 0,C 180,E1 -14667.591,E2 -14667.591} C_VEL
LIN {X 0,Y 334.244,Z 542.846,A -85,B 0,C 180,E1 -14670.002,E2 -14670.002} C_VEL
LIN {X 0,Y 334.104,Z 542.865,A -85,B 0,C 180,E1 -14672.413,E2 -14672.413} C_VEL
LIN {X 0,Y 334.012,Z 542.875,A -85,B 0,C 180,E1 -14676.041,E2 -14676.041} C_VEL
LIN {X 0,Y 333.983,Z 542.881,A -85,B 0,C 180,E1 -14678.503,E2 -14678.503} C_VEL
LIN {X 0,Y 333.79,Z 542.903,A -85,B 0,C 180,E1 -14682.156,E2 -14682.156} C_VEL
LIN {X 0,Y 333.777,Z 542.905,A -85,B 0,C 180,E1 -14685.888,E2 -14685.888} C_VEL
LIN {X 0,Y 333.795,Z 542.904,A -85,B 0,C 180,E1 -14688.656,E2 -14688.656} C_VEL
LIN {X 0,Y 333.692,Z 542.915,A -85,B 0,C 180,E1 -14692.28,E2 -14692.28} C_VEL
LIN {X 0,Y 333.736,Z 542.91,A -85,B 0,C 180,E1 -14696.248,E2 -14696.248} C_VEL
LIN {X 0,Y 333.686,Z 542.918,A -85,B 0,C 180,E1 -14698.82,E2 -14698.82} C_VEL
LIN {X 0,Y 333.04,Z 543.004,A -85,B 0,C 180,E1 -14699.826,E2 -14699.826} C_VEL
LIN {X 0,Y 330.189,Z 543.36,A -85,B 0,C 180,E1 -14701.464,E2 -14701.464} C_VEL
LIN {X 0,Y 327.752,Z 543.659,A -85,B 0,C 180,E1 -14702.79,E2 -14702.79} C_VEL
LIN {X 0,Y 326.694,Z 543.789,A -85,B 0,C 180,E1 -14703.817,E2 -14703.817} C_VEL
LIN {X 0,Y 326.603,Z 543.798,A -85,B 0,C 180,E1 -14704.165,E2 -14704.165} C_VEL
LIN {X 0,Y 326.629,Z 543.801,A -85,B 0,C 180,E1 -14707.24,E2 -14707.24} C_VEL
LIN {X 0,Y 326.581,Z 543.805,A -85,B 0,C 180,E1 -14711.133,E2 -14711.133} C_VEL
LIN {X 0,Y 326.559,Z 543.805,A -85,B 0,C 180,E1 -14714.749,E2 -14714.749} C_VEL
LIN {X 0,Y 326.58,Z 543.801,A -85,B 0,C 180,E1 -14718.156,E2 -14718.156} C_VEL
LIN {X 0,Y 326.627,Z 543.8,A -85,B 0,C 180,E1 -14721.393,E2 -14721.393} C_VEL
LIN {X 0,Y 326.623,Z 543.797,A -85,B 0,C 180,E1 -14724.853,E2 -14724.853} C_VEL
LIN {X 0,Y 326.612,Z 543.803,A -85,B 0,C 180,E1 -14727.457,E2 -14727.457} C_VEL
LIN {X 0,Y 326.666,Z 543.79,A -85,B 0,C 180,E1 -14730.342,E2 -14730.342} C_VEL
LIN {X 0,Y 326.695,Z 543.787,A -85,B 0,C 180,E1 -14734.517,E2 -14734.517} C_VEL
LIN {X 0,Y 326.624,Z 543.796,A -85,B 0,C 180,E1 -14738.544,E2 -14738.544} C_VEL
LIN {X 0,Y 326.713,Z 543.786,A -85,B 0,C 180,E1 -14741.176,E2 -14741.176} C_VEL
LIN {X 0,Y 326.77,Z 543.781,A -85,B 0,C 180,E1 -14745.434,E2 -14745.434} C_VEL
LIN {X 0,Y 326.777,Z 543.777,A -85,B 0,C 180,E1 -14748.84,E2 -14748.84} C_VEL
LIN {X 0,Y 326.965,Z 543.753,A -85,B 0,C 180,E1 -14752.591,E2 -14752.591} C_VEL
LIN {X 0,Y 326.782,Z 543.776,A -85,B 0,C 180,E1 -14755.066,E2 -14755.066} C_VEL
LIN {X 0,Y 327.053,Z 543.746,A -85,B 0,C 180,E1 -14757.537,E2 -14757.537} C_VEL
LIN {X 0,Y 327.205,Z 543.728,A -85,B 0,C 180,E1 -14760.001,E2 -14760.001} C_VEL
LIN {X 0,Y 327.053,Z 543.743,A -85,B 0,C 180,E1 -14762.464,E2 -14762.464} C_VEL
LIN {X 0,Y 327.004,Z 543.752,A -85,B 0,C 180,E1 -14766.17,E2 -14766.17} C_VEL
LIN {X 0,Y 326.923,Z 543.759,A -85,B 0,C 180,E1 -14768.655,E2 -14768.655} C_VEL
LIN {X 0,Y 326.742,Z 543.782,A -85,B 0,C 180,E1 -14772.422,E2 -14772.422} C_VEL
LIN {X 0,Y 326.763,Z 543.778,A -85,B 0,C 180,E1 -14774.958,E2 -14774.958} C_VEL
LIN {X 0,Y 326.741,Z 543.781,A -85,B 0,C 180,E1 -14778.838,E2 -14778.838} C_VEL
LIN {X 0,Y 326.611,Z 543.796,A -85,B 0,C 180,E1 -14782.789,E2 -14782.789} C_VEL
LIN {X 0,Y 326.698,Z 543.786,A -85,B 0,C 180,E1 -14785.484,E2 -14785.484} C_VEL
LIN {X 0,Y 326.656,Z 543.794,A -85,B 0,C 180,E1 -14789.66,E2 -14789.66} C_VEL
LIN {X 0,Y 326.615,Z 543.801,A -85,B 0,C 180,E1 -14794.019,E2 -14794.019} C_VEL
LIN {X 0,Y 326.635,Z 543.794,A -85,B 0,C 180,E1 -14797.238,E2 -14797.238} C_VEL
LIN {X 0,Y 326.585,Z 543.801,A -85,B 0,C 180,E1 -14801.131,E2 -14801.131} C_VEL
LIN {X 0,Y 326.535,Z 543.808,A -85,B 0,C 180,E1 -14804.742,E2 -14804.742} C_VEL
LIN {X 0,Y 326.584,Z 543.805,A -85,B 0,C 180,E1 -14808.154,E2 -14808.154} C_VEL
LIN {X 0,Y 326.632,Z 543.795,A -85,B 0,C 180,E1 -14811.391,E2 -14811.391} C_VEL
LIN {X 0,Y 326.628,Z 543.798,A -85,B 0,C 180,E1 -14814.85,E2 -14814.85} C_VEL
LIN {X 0,Y 326.652,Z 543.881,A -85,B 0,C 180,E1 -14818.684,E2 -14818.684} C_VEL
LIN {X 0,Y 329.068,Z 555.043,A -85,B 0,C 180,E1 -14821.973,E2 -14821.973} C_VEL
LIN {X 0,Y 330.727,Z 564.031,A -85,B 0,C 180,E1 -14824.511,E2 -14824.511} C_VEL
LIN {X 0,Y 330.183,Z 570.45,A -85,B 0,C 180,E1 -14826.177,E2 -14826.177} C_VEL
LIN {X 0,Y 335.922,Z 608.208,A -85,B 0,C 180,E1 -14827.471,E2 -14827.471} C_VEL
LIN {X 0,Y 334.301,Z 678.649,A -85,B 0,C 180,E1 -14829.099,E2 -14829.099} C_VEL
LIN {X 0,Y 333.519,Z 692.355,A -85,B 0,C 180,E1 -14829.652,E2 -14829.652} C_VEL
LIN {X 0,Y 332.536,Z 704.803,A -85,B 0,C 180,E1 -14830.395,E2 -14830.395} C_VEL
LIN {X 0,Y 331.514,Z 715.977,A -85,B 0,C 180,E1 -14831.296,E2 -14831.296} C_VEL
LIN {X 0,Y 330.205,Z 727.612,A -85,B 0,C 180,E1 -14832.503,E2 -14832.503} C_VEL
LIN {X 0,Y 329.057,Z 738.119,A -85,B 0,C 180,E1 -14833.878,E2 -14833.878} C_VEL
LIN {X 0,Y 327.98,Z 747.561,A -85,B 0,C 180,E1 -14835.415,E2 -14835.415} C_VEL
LIN {X 0,Y 326.874,Z 756.682,A -85,B 0,C 180,E1 -14837.267,E2 -14837.267} C_VEL
LIN {X 0,Y 326.051,Z 764.024,A -85,B 0,C 180,E1 -14839.127,E2 -14839.127} C_VEL
LIN {X 0,Y 325.553,Z 768.969,A -85,B 0,C 180,E1 -14840.681,E2 -14840.681} C_VEL
LIN {X 0,Y 325.179,Z 773.76,A -85,B 0,C 180,E1 -14842.547,E2 -14842.547} C_VEL
LIN {X 0,Y 324.958,Z 777.023,A -85,B 0,C 180,E1 -14844.194,E2 -14844.194} C_VEL
LIN {X 0,Y 324.907,Z 780.006,A -85,B 0,C 180,E1 -14846.278,E2 -14846.278} C_VEL
LIN {X 0,Y 324.84,Z 781.217,A -85,B 0,C 180,E1 -14847.518,E2 -14847.518} C_VEL
LIN {X 0,Y 324.835,Z 781.976,A -85,B 0,C 180,E1 -14848.759,E2 -14848.759} C_VEL
LIN {X 0,Y 324.875,Z 782.325,A -85,B 0,C 180,E1 -14849.998,E2 -14849.998} C_VEL
LIN {X 0,Y 324.822,Z 782.277,A -85,B 0,C 180,E1 -14851.238,E2 -14851.238} C_VEL
LIN {X 0,Y 324.836,Z 781.834,A -85,B 0,C 180,E1 -14852.478,E2 -14852.478} C_VEL
LIN {X 0,Y 324.882,Z 780.949,A -85,B 0,C 180,E1 -14853.719,E2 -14853.719} C_VEL
LIN {X 0,Y 324.915,Z 778.647,A -85,B 0,C 180,E1 -14855.731,E2 -14855.731} C_VEL
LIN {X 0,Y 325.289,Z 774.523,A -85,B 0,C 180,E1 -14858.071,E2 -14858.071} C_VEL
LIN {X 0,Y 325.797,Z 770.022,A -85,B 0,C 180,E1 -14859.936,E2 -14859.936} C_VEL
LIN {X 0,Y 326.533,Z 764.317,A -85,B 0,C 180,E1 -14861.797,E2 -14861.797} C_VEL
LIN {X 0,Y 327.651,Z 757.202,A -85,B 0,C 180,E1 -14863.645,E2 -14863.645} C_VEL
LIN {X 0,Y 328.987,Z 748.338,A -85,B 0,C 180,E1 -14865.486,E2 -14865.486} C_VEL
LIN {X 0,Y 330.422,Z 738.401,A -85,B 0,C 180,E1 -14867.147,E2 -14867.147} C_VEL
LIN {X 0,Y 331.871,Z 728.091,A -85,B 0,C 180,E1 -14868.519,E2 -14868.519} C_VEL
LIN {X 0,Y 333.347,Z 716.815,A -85,B 0,C 180,E1 -14869.712,E2 -14869.712} C_VEL
LIN {X 0,Y 334.75,Z 704.186,A -85,B 0,C 180,E1 -14870.748,E2 -14870.748} C_VEL
LIN {X 0,Y 335.876,Z 691.945,A -85,B 0,C 180,E1 -14871.478,E2 -14871.478} C_VEL
LIN {X 0,Y 336.764,Z 678.646,A -85,B 0,C 180,E1 -14872.022,E2 -14872.022} C_VEL
LIN {X 0,Y 338.642,Z 613.151,A -85,B 0,C 180,E1 -14873.569,E2 -14873.569} C_VEL
LIN {X 0,Y 338.568,Z 606.893,A -85,B 0,C 180,E1 -14873.736,E2 -14873.736} C_VEL
LIN {X 0,Y 335.055,Z 585.384,A -85,B 0,C 180,E1 -14874.614,E2 -14874.614} C_VEL
LIN {X 0,Y 331.692,Z 569.161,A -85,B 0,C 180,E1 -14875.406,E2 -14875.406} C_VEL
LIN {X 0,Y 331.44,Z 565.559,A -85,B 0,C 180,E1 -14876.44,E2 -14876.44} C_VEL
LIN {X 0,Y 329.601,Z 556.08,A -85,B 0,C 180,E1 -14879.366,E2 -14879.366} C_VEL
LIN {X 0,Y 327.31,Z 546.762,A -85,B 0,C 180,E1 -14882.464,E2 -14882.464} C_VEL
LIN {X 0,Y 326.594,Z 543.805,A -85,B 0,C 180,E1 -14883.569,E2 -14883.569} C_VEL
LIN {X 0,Y 326.627,Z 543.802,A -85,B 0,C 180,E1 -14887.237,E2 -14887.237} C_VEL
LIN {X 0,Y 326.599,Z 543.806,A -85,B 0,C 180,E1 -14890.205,E2 -14890.205} C_VEL
LIN {X 0,Y 326.58,Z 543.813,A -85,B 0,C 180,E1 -14893.52,E2 -14893.52} C_VEL
LIN {X 0,Y 326.596,Z 543.803,A -85,B 0,C 180,E1 -14897.021,E2 -14897.021} C_VEL
LIN {X 0,Y 326.627,Z 543.797,A -85,B 0,C 180,E1 -14900.766,E2 -14900.766} C_VEL
LIN {X 0,Y 326.605,Z 543.801,A -85,B 0,C 180,E1 -14904.479,E2 -14904.479} C_VEL
LIN {X 0,Y 326.599,Z 543.805,A -85,B 0,C 180,E1 -14907.454,E2 -14907.454} C_VEL
LIN {X 0,Y 326.652,Z 543.794,A -85,B 0,C 180,E1 -14910.339,E2 -14910.339} C_VEL
LIN {X 0,Y 326.681,Z 543.791,A -85,B 0,C 180,E1 -14914.515,E2 -14914.515} C_VEL
LIN {X 0,Y 326.637,Z 543.797,A -85,B 0,C 180,E1 -14918.544,E2 -14918.544} C_VEL
LIN {X 0,Y 326.734,Z 543.778,A -85,B 0,C 180,E1 -14921.176,E2 -14921.176} C_VEL
LIN {X 0,Y 326.752,Z 543.78,A -85,B 0,C 180,E1 -14925.432,E2 -14925.432} C_VEL
LIN {X 0,Y 326.763,Z 543.775,A -85,B 0,C 180,E1 -14928.838,E2 -14928.838} C_VEL
LIN {X 0,Y 326.968,Z 543.751,A -85,B 0,C 180,E1 -14932.589,E2 -14932.589} C_VEL
LIN {X 0,Y 326.77,Z 543.777,A -85,B 0,C 180,E1 -14935.064,E2 -14935.064} C_VEL
LIN {X 0,Y 327.058,Z 543.745,A -85,B 0,C 180,E1 -14937.536,E2 -14937.536} C_VEL
LIN {X 0,Y 327.207,Z 543.727,A -85,B 0,C 180,E1 -14939.999,E2 -14939.999} C_VEL
LIN {X 0,Y 327.058,Z 543.742,A -85,B 0,C 180,E1 -14942.463,E2 -14942.463} C_VEL
LIN {X 0,Y 326.963,Z 543.754,A -85,B 0,C 180,E1 -14946.648,E2 -14946.648} C_VEL
LIN {X 0,Y 326.804,Z 543.775,A -85,B 0,C 180,E1 -14949.906,E2 -14949.906} C_VEL
LIN {X 0,Y 326.748,Z 543.785,A -85,B 0,C 180,E1 -14953.685,E2 -14953.685} C_VEL
LIN {X 0,Y 326.687,Z 543.795,A -85,B 0,C 180,E1 -14957.528,E2 -14957.528} C_VEL
LIN {X 0,Y 326.655,Z 543.825,A -85,B 0,C 180,E1 -14960.628,E2 -14960.628} C_VEL
LIN {X 0,Y 328.675,Z 552.882,A -85,B 0,C 180,E1 -14963.97,E2 -14963.97} C_VEL
LIN {X 0,Y 329.027,Z 554.376,A -85,B 0,C 180,E1 -14964.446,E2 -14964.446} C_VEL
LIN {X 0,Y 336.68,Z 571.806,A -85,B 0,C 180,E1 -14965.652,E2 -14965.652} C_VEL
LIN {X 0,Y 338.417,Z 578.97,A -85,B 0,C 180,E1 -14965.999,E2 -14965.999} C_VEL
LIN {X 0,Y 339.333,Z 584.854,A -85,B 0,C 180,E1 -14966.235,E2 -14966.235} C_VEL
LIN {X 0,Y 337.022,Z 661.479,A -85,B 0,C 180,E1 -14968.04,E2 -14968.04} C_VEL
LIN {X 0,Y 336.226,Z 675.163,A -85,B 0,C 180,E1 -14968.613,E2 -14968.613} C_VEL
LIN {X 0,Y 335.306,Z 686.94,A -85,B 0,C 180,E1 -14969.336,E2 -14969.336} C_VEL
LIN {X 0,Y 334.048,Z 698.964,A -85,B 0,C 180,E1 -14970.326,E2 -14970.326} C_VEL
LIN {X 0,Y 332.7,Z 710.19,A -85,B 0,C 180,E1 -14971.521,E2 -14971.521} C_VEL
LIN {X 0,Y 331.246,Z 721.019,A -85,B 0,C 180,E1 -14972.976,E2 -14972.976} C_VEL
LIN {X 0,Y 329.828,Z 730.117,A -85,B 0,C 180,E1 -14974.501,E2 -14974.501} C_VEL
LIN {X 0,Y 328.497,Z 738.49,A -85,B 0,C 180,E1 -14976.235,E2 -14976.235} C_VEL
LIN {X 0,Y 327.441,Z 745.235,A -85,B 0,C 180,E1 -14977.964,E2 -14977.964} C_VEL
LIN {X 0,Y 326.555,Z 750.727,A -85,B 0,C 180,E1 -14979.705,E2 -14979.705} C_VEL
LIN {X 0,Y 325.787,Z 756.225,A -85,B 0,C 180,E1 -14981.969,E2 -14981.969} C_VEL
LIN {X 0,Y 325.322,Z 759.402,A -85,B 0,C 180,E1 -14983.732,E2 -14983.732} C_VEL
LIN {X 0,Y 324.846,Z 762.31,A -85,B 0,C 180,E1 -14986.189,E2 -14986.189} C_VEL
LIN {X 0,Y 324.689,Z 763.368,A -85,B 0,C 180,E1 -14987.858,E2 -14987.858} C_VEL
LIN {X 0,Y 324.606,Z 763.716,A -85,B 0,C 180,E1 -14989.497,E2 -14989.497} C_VEL
LIN {X 0,Y 324.589,Z 763.285,A -85,B 0,C 180,E1 -14991.211,E2 -14991.211} C_VEL
LIN {X 0,Y 324.737,Z 761.835,A -85,B 0,C 180,E1 -14993.201,E2 -14993.201} C_VEL
LIN {X 0,Y 325.021,Z 759.22,A -85,B 0,C 180,E1 -14995.252,E2 -14995.252} C_VEL
LIN {X 0,Y 325.414,Z 755.205,A -85,B 0,C 180,E1 -14997.381,E2 -14997.381} C_VEL
LIN {X 0,Y 326.032,Z 749.519,A -85,B 0,C 180,E1 -14999.568,E2 -14999.568} C_VEL
LIN {X 0,Y 326.742,Z 743.364,A -85,B 0,C 180,E1 -15001.409,E2 -15001.409} C_VEL
LIN {X 0,Y 327.667,Z 735.775,A -85,B 0,C 180,E1 -15003.232,E2 -15003.232} C_VEL
LIN {X 0,Y 328.843,Z 726.306,A -85,B 0,C 180,E1 -15005.035,E2 -15005.035} C_VEL
LIN {X 0,Y 330.025,Z 716.059,A -85,B 0,C 180,E1 -15006.604,E2 -15006.604} C_VEL
LIN {X 0,Y 331.141,Z 705.959,A -85,B 0,C 180,E1 -15007.843,E2 -15007.843} C_VEL
LIN {X 0,Y 332.224,Z 693.975,A -85,B 0,C 180,E1 -15009.006,E2 -15009.006} C_VEL
LIN {X 0,Y 333.297,Z 680.944,A -85,B 0,C 180,E1 -15009.963,E2 -15009.963} C_VEL
LIN {X 0,Y 334.093,Z 667.666,A -85,B 0,C 180,E1 -15010.646,E2 -15010.646} C_VEL
LIN {X 0,Y 334.576,Z 654.637,A -85,B 0,C 180,E1 -15011.074,E2 -15011.074} C_VEL
LIN {X 0,Y 336.22,Z 582.019,A -85,B 0,C 180,E1 -15012.729,E2 -15012.729} C_VEL
LIN {X 0,Y 332.859,Z 565.366,A -85,B 0,C 180,E1 -15013.352,E2 -15013.352} C_VEL
LIN {X 0,Y 328.486,Z 552.821,A -85,B 0,C 180,E1 -15013.967,E2 -15013.967} C_VEL
LIN {X 0,Y 326.766,Z 543.784,A -85,B 0,C 180,E1 -15016.911,E2 -15016.911} C_VEL
LIN {X 0,Y 326.921,Z 543.76,A -85,B 0,C 180,E1 -15021.445,E2 -15021.445} C_VEL
LIN {X 0,Y 326.986,Z 543.751,A -85,B 0,C 180,E1 -15023.833,E2 -15023.833} C_VEL
LIN {X 0,Y 327.045,Z 543.744,A -85,B 0,C 180,E1 -15027.539,E2 -15027.539} C_VEL
LIN {X 0,Y 327.196,Z 543.725,A -85,B 0,C 180,E1 -15030.002,E2 -15030.002} C_VEL
LIN {X 0,Y 327.045,Z 543.745,A -85,B 0,C 180,E1 -15032.465,E2 -15032.465} C_VEL
LIN {X 0,Y 326.987,Z 543.75,A -85,B 0,C 180,E1 -15036.171,E2 -15036.171} C_VEL
LIN {X 0,Y 326.913,Z 543.763,A -85,B 0,C 180,E1 -15038.657,E2 -15038.657} C_VEL
LIN {X 0,Y 326.733,Z 543.782,A -85,B 0,C 180,E1 -15042.423,E2 -15042.423} C_VEL
LIN {X 0,Y 326.753,Z 543.784,A -85,B 0,C 180,E1 -15044.959,E2 -15044.959} C_VEL
LIN {X 0,Y 326.732,Z 543.786,A -85,B 0,C 180,E1 -15048.84,E2 -15048.84} C_VEL
LIN {X 0,Y 326.621,Z 543.797,A -85,B 0,C 180,E1 -15052.789,E2 -15052.789} C_VEL
LIN {X 0,Y 326.691,Z 543.79,A -85,B 0,C 180,E1 -15055.485,E2 -15055.485} C_VEL
LIN {X 0,Y 326.649,Z 543.795,A -85,B 0,C 180,E1 -15059.662,E2 -15059.662} C_VEL
LIN {X 0,Y 326.608,Z 543.798,A -85,B 0,C 180,E1 -15064.021,E2 -15064.021} C_VEL
LIN {X 0,Y 326.603,Z 543.798,A -85,B 0,C 180,E1 -15064.165,E2 -15064.165} C_VEL
LIN {X 0,Y 325.872,Z 543.895,A -85,B 0,C 180,E1 -15065.196,E2 -15065.196} C_VEL
LIN {X 0,Y 322.859,Z 544.272,A -85,B 0,C 180,E1 -15066.87,E2 -15066.87} C_VEL
LIN {X 0,Y 320.43,Z 544.576,A -85,B 0,C 180,E1 -15068.228,E2 -15068.228} C_VEL
LIN {X 0,Y 319.542,Z 544.684,A -85,B 0,C 180,E1 -15069.281,E2 -15069.281} C_VEL
LIN {X 0,Y 319.551,Z 544.679,A -85,B 0,C 180,E1 -15069.636,E2 -15069.636} C_VEL
LIN {X 0,Y 319.559,Z 544.681,A -85,B 0,C 180,E1 -15073.469,E2 -15073.469} C_VEL
LIN {X 0,Y 319.565,Z 544.678,A -85,B 0,C 180,E1 -15077.019,E2 -15077.019} C_VEL
LIN {X 0,Y 319.55,Z 544.675,A -85,B 0,C 180,E1 -15080.372,E2 -15080.372} C_VEL
LIN {X 0,Y 319.563,Z 544.68,A -85,B 0,C 180,E1 -15083.574,E2 -15083.574} C_VEL
LIN {X 0,Y 319.582,Z 544.673,A -85,B 0,C 180,E1 -15086.688,E2 -15086.688} C_VEL
LIN {X 0,Y 319.596,Z 544.675,A -85,B 0,C 180,E1 -15089.618,E2 -15089.618} C_VEL
LIN {X 0,Y 319.614,Z 544.668,A -85,B 0,C 180,E1 -15092.499,E2 -15092.499} C_VEL
LIN {X 0,Y 319.609,Z 544.673,A -85,B 0,C 180,E1 -15095.305,E2 -15095.305} C_VEL
LIN {X 0,Y 319.592,Z 544.675,A -85,B 0,C 180,E1 -15099.4,E2 -15099.4} C_VEL
LIN {X 0,Y 319.63,Z 544.667,A -85,B 0,C 180,E1 -15102.072,E2 -15102.072} C_VEL
LIN {X 0,Y 319.739,Z 544.656,A -85,B 0,C 180,E1 -15106.009,E2 -15106.009} C_VEL
LIN {X 0,Y 319.76,Z 544.655,A -85,B 0,C 180,E1 -15109.874,E2 -15109.874} C_VEL
LIN {X 0,Y 319.92,Z 544.63,A -85,B 0,C 180,E1 -15112.427,E2 -15112.427} C_VEL
LIN {X 0,Y 319.751,Z 544.651,A -85,B 0,C 180,E1 -15114.957,E2 -15114.957} C_VEL
LIN {X 0,Y 319.997,Z 544.624,A -85,B 0,C 180,E1 -15117.483,E2 -15117.483} C_VEL
LIN {X 0,Y 320.156,Z 544.606,A -85,B 0,C 180,E1 -15120.001,E2 -15120.001} C_VEL
LIN {X 0,Y 319.997,Z 544.621,A -85,B 0,C 180,E1 -15122.518,E2 -15122.518} C_VEL
LIN {X 0,Y 319.96,Z 544.628,A -85,B 0,C 180,E1 -15126.306,E2 -15126.306} C_VEL
LIN {X 0,Y 319.851,Z 544.64,A -85,B 0,C 180,E1 -15128.848,E2 -15128.848} C_VEL
LIN {X 0,Y 319.69,Z 544.659,A -85,B 0,C 180,E1 -15132.7,E2 -15132.7} C_VEL
LIN {X 0,Y 319.708,Z 544.658,A -85,B 0,C 180,E1 -15135.296,E2 -15135.296} C_VEL
LIN {X 0,Y 319.66,Z 544.664,A -85,B 0,C 180,E1 -15139.257,E2 -15139.257} C_VEL
LIN {X 0,Y 319.569,Z 544.672,A -85,B 0,C 180,E1 -15143.32,E2 -15143.32} C_VEL
LIN {X 0,Y 319.643,Z 544.669,A -85,B 0,C 180,E1 -15146.088,E2 -15146.088} C_VEL
LIN {X 0,Y 319.588,Z 544.672,A -85,B 0,C 180,E1 -15148.934,E2 -15148.934} C_VEL
LIN {X 0,Y 319.539,Z 544.682,A -85,B 0,C 180,E1 -15151.862,E2 -15151.862} C_VEL
LIN {X 0,Y 319.588,Z 544.673,A -85,B 0,C 180,E1 -15155.542,E2 -15155.542} C_VEL
LIN {X 0,Y 319.581,Z 544.677,A -85,B 0,C 180,E1 -15158.008,E2 -15158.008} C_VEL
LIN {X 0,Y 319.533,Z 544.68,A -85,B 0,C 180,E1 -15161.596,E2 -15161.596} C_VEL
LIN {X 0,Y 319.496,Z 544.683,A -85,B 0,C 180,E1 -15165.257,E2 -15165.257} C_VEL
LIN {X 0,Y 319.536,Z 544.681,A -85,B 0,C 180,E1 -15168.711,E2 -15168.711} C_VEL
LIN {X 0,Y 319.586,Z 544.678,A -85,B 0,C 180,E1 -15172.343,E2 -15172.343} C_VEL
LIN {X 0,Y 319.568,Z 544.676,A -85,B 0,C 180,E1 -15175.123,E2 -15175.123} C_VEL
LIN {X 0,Y 319.589,Z 544.763,A -85,B 0,C 180,E1 -15178.319,E2 -15178.319} C_VEL
LIN {X 0,Y 322.247,Z 557.096,A -85,B 0,C 180,E1 -15182.035,E2 -15182.035} C_VEL
LIN {X 0,Y 323.811,Z 566.097,A -85,B 0,C 180,E1 -15184.616,E2 -15184.616} C_VEL
LIN {X 0,Y 323.37,Z 570.473,A -85,B 0,C 180,E1 -15185.722,E2 -15185.722} C_VEL
LIN {X 0,Y 329.222,Z 609.132,A -85,B 0,C 180,E1 -15187.083,E2 -15187.083} C_VEL
LIN {X 0,Y 327.551,Z 678.706,A -85,B 0,C 180,E1 -15188.73,E2 -15188.73} C_VEL
LIN {X 0,Y 326.743,Z 692.318,A -85,B 0,C 180,E1 -15189.293,E2 -15189.293} C_VEL
LIN {X 0,Y 325.728,Z 704.717,A -85,B 0,C 180,E1 -15190.05,E2 -15190.05} C_VEL
LIN {X 0,Y 324.597,Z 716.655,A -85,B 0,C 180,E1 -15191.047,E2 -15191.047} C_VEL
LIN {X 0,Y 323.257,Z 728.132,A -85,B 0,C 180,E1 -15192.278,E2 -15192.278} C_VEL
LIN {X 0,Y 322.049,Z 738.581,A -85,B 0,C 180,E1 -15193.692,E2 -15193.692} C_VEL
LIN {X 0,Y 321.094,Z 746.995,A -85,B 0,C 180,E1 -15195.095,E2 -15195.095} C_VEL
LIN {X 0,Y 319.891,Z 756.178,A -85,B 0,C 180,E1 -15196.984,E2 -15196.984} C_VEL
LIN {X 0,Y 319.009,Z 763.573,A -85,B 0,C 180,E1 -15198.884,E2 -15198.884} C_VEL
LIN {X 0,Y 318.502,Z 768.568,A -85,B 0,C 180,E1 -15200.472,E2 -15200.472} C_VEL
LIN {X 0,Y 318.098,Z 773.403,A -85,B 0,C 180,E1 -15202.381,E2 -15202.381} C_VEL
LIN {X 0,Y 317.852,Z 777.051,A -85,B 0,C 180,E1 -15204.268,E2 -15204.268} C_VEL
LIN {X 0,Y 317.815,Z 779.725,A -85,B 0,C 180,E1 -15206.194,E2 -15206.194} C_VEL
LIN {X 0,Y 317.762,Z 780.956,A -85,B 0,C 180,E1 -15207.463,E2 -15207.463} C_VEL
LIN {X 0,Y 317.746,Z 781.746,A -85,B 0,C 180,E1 -15208.731,E2 -15208.731} C_VEL
LIN {X 0,Y 317.783,Z 782.111,A -85,B 0,C 180,E1 -15209.998,E2 -15209.998} C_VEL
LIN {X 0,Y 317.735,Z 782.077,A -85,B 0,C 180,E1 -15211.266,E2 -15211.266} C_VEL
LIN {X 0,Y 317.757,Z 781.651,A -85,B 0,C 180,E1 -15212.533,E2 -15212.533} C_VEL
LIN {X 0,Y 317.791,Z 780.794,A -85,B 0,C 180,E1 -15213.802,E2 -15213.802} C_VEL
LIN {X 0,Y 317.832,Z 778.756,A -85,B 0,C 180,E1 -15215.696,E2 -15215.696} C_VEL
LIN {X 0,Y 318.086,Z 775.695,A -85,B 0,C 180,E1 -15217.616,E2 -15217.616} C_VEL
LIN {X 0,Y 318.58,Z 771.606,A -85,B 0,C 180,E1 -15219.522,E2 -15219.522} C_VEL
LIN {X 0,Y 319.424,Z 765.339,A -85,B 0,C 180,E1 -15221.741,E2 -15221.741} C_VEL
LIN {X 0,Y 320.541,Z 758.53,A -85,B 0,C 180,E1 -15223.631,E2 -15223.631} C_VEL
LIN {X 0,Y 321.941,Z 750.099,A -85,B 0,C 180,E1 -15225.509,E2 -15225.509} C_VEL
LIN {X 0,Y 323.192,Z 741.448,A -85,B 0,C 180,E1 -15227.069,E2 -15227.069} C_VEL
LIN {X 0,Y 324.803,Z 730.809,A -85,B 0,C 180,E1 -15228.61,E2 -15228.61} C_VEL
LIN {X 0,Y 326.256,Z 720.302,A -85,B 0,C 180,E1 -15229.831,E2 -15229.831} C_VEL
LIN {X 0,Y 327.765,Z 708.738,A -85,B 0,C 180,E1 -15230.882,E2 -15230.882} C_VEL
LIN {X 0,Y 329.031,Z 695.596,A -85,B 0,C 180,E1 -15231.783,E2 -15231.783} C_VEL
LIN {X 0,Y 330.094,Z 682.468,A -85,B 0,C 180,E1 -15232.408,E2 -15232.408} C_VEL
LIN {X 0,Y 330.753,Z 668.031,A -85,B 0,C 180,E1 -15232.823,E2 -15232.823} C_VEL
LIN {X 0,Y 332.376,Z 608.895,A -85,B 0,C 180,E1 -15234.234,E2 -15234.234} C_VEL
LIN {X 0,Y 329.102,Z 588.188,A -85,B 0,C 180,E1 -15235.098,E2 -15235.098} C_VEL
LIN {X 0,Y 325.494,Z 571.205,A -85,B 0,C 180,E1 -15235.921,E2 -15235.921} C_VEL
LIN {X 0,Y 324.857,Z 569.004,A -85,B 0,C 180,E1 -15236.067,E2 -15236.067} C_VEL
LIN {X 0,Y 322.86,Z 558.223,A -85,B 0,C 180,E1 -15239.457,E2 -15239.457} C_VEL
LIN {X 0,Y 320.437,Z 548.233,A -85,B 0,C 180,E1 -15242.874,E2 -15242.874} C_VEL
LIN {X 0,Y 319.557,Z 544.68,A -85,B 0,C 180,E1 -15244.204,E2 -15244.204} C_VEL
LIN {X 0,Y 319.594,Z 544.68,A -85,B 0,C 180,E1 -15248.002,E2 -15248.002} C_VEL
LIN {X 0,Y 319.564,Z 544.687,A -85,B 0,C 180,E1 -15251.604,E2 -15251.604} C_VEL
LIN {X 0,Y 319.503,Z 544.689,A -85,B 0,C 180,E1 -15255.259,E2 -15255.259} C_VEL
LIN {X 0,Y 319.538,Z 544.683,A -85,B 0,C 180,E1 -15258.713,E2 -15258.713} C_VEL
LIN {X 0,Y 319.575,Z 544.673,A -85,B 0,C 180,E1 -15262.341,E2 -15262.341} C_VEL
LIN {X 0,Y 319.553,Z 544.678,A -85,B 0,C 180,E1 -15265.122,E2 -15265.122} C_VEL
LIN {X 0,Y 319.562,Z 544.673,A -85,B 0,C 180,E1 -15269.056,E2 -15269.056} C_VEL
LIN {X 0,Y 319.6,Z 544.667,A -85,B 0,C 180,E1 -15272.497,E2 -15272.497} C_VEL
LIN {X 0,Y 319.596,Z 544.674,A -85,B 0,C 180,E1 -15275.303,E2 -15275.303} C_VEL
LIN {X 0,Y 319.587,Z 544.676,A -85,B 0,C 180,E1 -15278.046,E2 -15278.046} C_VEL
LIN {X 0,Y 319.679,Z 544.655,A -85,B 0,C 180,E1 -15280.961,E2 -15280.961} C_VEL
LIN {X 0,Y 319.72,Z 544.654,A -85,B 0,C 180,E1 -15285.275,E2 -15285.275} C_VEL
LIN {X 0,Y 319.749,Z 544.656,A -85,B 0,C 180,E1 -15289.872,E2 -15289.872} C_VEL
LIN {X 0,Y 319.922,Z 544.629,A -85,B 0,C 180,E1 -15292.425,E2 -15292.425} C_VEL
LIN {X 0,Y 319.739,Z 544.653,A -85,B 0,C 180,E1 -15294.955,E2 -15294.955} C_VEL
LIN {X 0,Y 319.998,Z 544.625,A -85,B 0,C 180,E1 -15297.482,E2 -15297.482} C_VEL
LIN {X 0,Y 320.158,Z 544.606,A -85,B 0,C 180,E1 -15299.999,E2 -15299.999} C_VEL
LIN {X 0,Y 319.999,Z 544.622,A -85,B 0,C 180,E1 -15302.517,E2 -15302.517} C_VEL
LIN {X 0,Y 319.923,Z 544.632,A -85,B 0,C 180,E1 -15306.637,E2 -15306.637} C_VEL
LIN {X 0,Y 319.748,Z 544.655,A -85,B 0,C 180,E1 -15310.127,E2 -15310.127} C_VEL
LIN {X 0,Y 319.719,Z 544.664,A -85,B 0,C 180,E1 -15314.724,E2 -15314.724} C_VEL
LIN {X 0,Y 319.666,Z 544.669,A -85,B 0,C 180,E1 -15319.033,E2 -15319.033} C_VEL
LIN {X 0,Y 319.643,Z 544.765,A -85,B 0,C 180,E1 -15320.009,E2 -15320.009} C_VEL
LIN {X 0,Y 321.667,Z 553.701,A -85,B 0,C 180,E1 -15323.421,E2 -15323.421} C_VEL
LIN {X 0,Y 321.839,Z 554.51,A -85,B 0,C 180,E1 -15323.698,E2 -15323.698} C_VEL
LIN {X 0,Y 329.461,Z 571.41,A -85,B 0,C 180,E1 -15324.958,E2 -15324.958} C_VEL
LIN {X 0,Y 331.427,Z 576.681,A -85,B 0,C 180,E1 -15325.29,E2 -15325.29} C_VEL
LIN {X 0,Y 333.063,Z 585.65,A -85,B 0,C 180,E1 -15325.684,E2 -15325.684} C_VEL
LIN {X 0,Y 330.633,Z 661.885,A -85,B 0,C 180,E1 -15327.523,E2 -15327.523} C_VEL
LIN {X 0,Y 329.793,Z 675.353,A -85,B 0,C 180,E1 -15328.1,E2 -15328.1} C_VEL
LIN {X 0,Y 328.86,Z 686.838,A -85,B 0,C 180,E1 -15328.817,E2 -15328.817} C_VEL
LIN {X 0,Y 327.545,Z 698.941,A -85,B 0,C 180,E1 -15329.826,E2 -15329.826} C_VEL
LIN {X 0,Y 326.209,Z 709.736,A -85,B 0,C 180,E1 -15330.986,E2 -15330.986} C_VEL
LIN {X 0,Y 324.668,Z 720.393,A -85,B 0,C 180,E1 -15332.415,E2 -15332.415} C_VEL
LIN {X 0,Y 323.229,Z 729.463,A -85,B 0,C 180,E1 -15333.933,E2 -15333.933} C_VEL
LIN {X 0,Y 321.849,Z 737.754,A -85,B 0,C 180,E1 -15335.647,E2 -15335.647} C_VEL
LIN {X 0,Y 320.668,Z 744.755,A -85,B 0,C 180,E1 -15337.434,E2 -15337.434} C_VEL
LIN {X 0,Y 319.502,Z 751.573,A -85,B 0,C 180,E1 -15339.635,E2 -15339.635} C_VEL
LIN {X 0,Y 318.862,Z 755.924,A -85,B 0,C 180,E1 -15341.466,E2 -15341.466} C_VEL
LIN {X 0,Y 318.339,Z 759.16,A -85,B 0,C 180,E1 -15343.239,E2 -15343.239} C_VEL
LIN {X 0,Y 317.977,Z 761.519,A -85,B 0,C 180,E1 -15345.012,E2 -15345.012} C_VEL
LIN {X 0,Y 317.682,Z 763.133,A -85,B 0,C 180,E1 -15346.89,E2 -15346.89} C_VEL
LIN {X 0,Y 317.526,Z 763.863,A -85,B 0,C 180,E1 -15348.81,E2 -15348.81} C_VEL
LIN {X 0,Y 317.489,Z 763.65,A -85,B 0,C 180,E1 -15350.783,E2 -15350.783} C_VEL
LIN {X 0,Y 317.669,Z 761.935,A -85,B 0,C 180,E1 -15353.323,E2 -15353.323} C_VEL
LIN {X 0,Y 317.997,Z 758.786,A -85,B 0,C 180,E1 -15355.699,E2 -15355.699} C_VEL
LIN {X 0,Y 318.473,Z 754.166,A -85,B 0,C 180,E1 -15358.022,E2 -15358.022} C_VEL
LIN {X 0,Y 319.048,Z 749.099,A -85,B 0,C 180,E1 -15359.927,E2 -15359.927} C_VEL
LIN {X 0,Y 319.716,Z 743.704,A -85,B 0,C 180,E1 -15361.554,E2 -15361.554} C_VEL
LIN {X 0,Y 320.574,Z 736.808,A -85,B 0,C 180,E1 -15363.264,E2 -15363.264} C_VEL
LIN {X 0,Y 321.806,Z 727.384,A -85,B 0,C 180,E1 -15365.142,E2 -15365.142} C_VEL
LIN {X 0,Y 322.931,Z 717.68,A -85,B 0,C 180,E1 -15366.692,E2 -15366.692} C_VEL
LIN {X 0,Y 324.181,Z 707.186,A -85,B 0,C 180,E1 -15368.042,E2 -15368.042} C_VEL
LIN {X 0,Y 325.356,Z 694.847,A -85,B 0,C 180,E1 -15369.287,E2 -15369.287} C_VEL
LIN {X 0,Y 326.462,Z 681.843,A -85,B 0,C 180,E1 -15370.277,E2 -15370.277} C_VEL
LIN {X 0,Y 327.208,Z 669.305,A -85,B 0,C 180,E1 -15370.96,E2 -15370.96} C_VEL
LIN {X 0,Y 327.767,Z 656.324,A -85,B 0,C 180,E1 -15371.417,E2 -15371.417} C_VEL
LIN {X 0,Y 329.615,Z 583.209,A -85,B 0,C 180,E1 -15373.117,E2 -15373.117} C_VEL
LIN {X 0,Y 326.453,Z 567.607,A -85,B 0,C 180,E1 -15373.716,E2 -15373.716} C_VEL
LIN {X 0,Y 321.347,Z 552.978,A -85,B 0,C 180,E1 -15374.468,E2 -15374.468} C_VEL
LIN {X 0,Y 319.703,Z 544.664,A -85,B 0,C 180,E1 -15377.222,E2 -15377.222} C_VEL
LIN {X 0,Y 319.869,Z 544.639,A -85,B 0,C 180,E1 -15381.38,E2 -15381.38} C_VEL
LIN {X 0,Y 319.941,Z 544.629,A -85,B 0,C 180,E1 -15383.696,E2 -15383.696} C_VEL
LIN {X 0,Y 319.988,Z 544.624,A -85,B 0,C 180,E1 -15387.484,E2 -15387.484} C_VEL
LIN {X 0,Y 320.148,Z 544.603,A -85,B 0,C 180,E1 -15390.002,E2 -15390.002} C_VEL
LIN {X 0,Y 319.989,Z 544.624,A -85,B 0,C 180,E1 -15392.519,E2 -15392.519} C_VEL
LIN {X 0,Y 319.943,Z 544.628,A -85,B 0,C 180,E1 -15396.307,E2 -15396.307} C_VEL
LIN {X 0,Y 319.841,Z 544.645,A -85,B 0,C 180,E1 -15398.85,E2 -15398.85} C_VEL
LIN {X 0,Y 319.681,Z 544.662,A -85,B 0,C 180,E1 -15402.702,E2 -15402.702} C_VEL
LIN {X 0,Y 319.699,Z 544.662,A -85,B 0,C 180,E1 -15405.297,E2 -15405.297} C_VEL
LIN {X 0,Y 319.674,Z 544.665,A -85,B 0,C 180,E1 -15409.257,E2 -15409.257} C_VEL
LIN {X 0,Y 319.571,Z 544.677,A -85,B 0,C 180,E1 -15413.321,E2 -15413.321} C_VEL
LIN {X 0,Y 319.619,Z 544.668,A -85,B 0,C 180,E1 -15416.091,E2 -15416.091} C_VEL
LIN {X 0,Y 319.581,Z 544.677,A -85,B 0,C 180,E1 -15418.936,E2 -15418.936} C_VEL
LIN {X 0,Y 319.532,Z 544.679,A -85,B 0,C 180,E1 -15421.864,E2 -15421.864} C_VEL
LIN {X 0,Y 319.582,Z 544.677,A -85,B 0,C 180,E1 -15425.545,E2 -15425.545} C_VEL
LIN {X 0,Y 319.551,Z 544.679,A -85,B 0,C 180,E1 -15429.636,E2 -15429.636} C_VEL
LIN {X 0,Y 319.077,Z 544.737,A -85,B 0,C 180,E1 -15430.687,E2 -15430.687} C_VEL
LIN {X 0,Y 317.52,Z 544.932,A -85,B 0,C 180,E1 -15431.717,E2 -15431.717} C_VEL
LIN {X 0,Y 313.633,Z 545.416,A -85,B 0,C 180,E1 -15433.779,E2 -15433.779} C_VEL
LIN {X 0,Y 312.53,Z 545.553,A -85,B 0,C 180,E1 -15434.855,E2 -15434.855} C_VEL
LIN {X 0,Y 312.448,Z 545.56,A -85,B 0,C 180,E1 -15435.22,E2 -15435.22} C_VEL
LIN {X 0,Y 312.489,Z 545.557,A -85,B 0,C 180,E1 -15437.92,E2 -15437.92} C_VEL
LIN {X 0,Y 312.509,Z 545.555,A -85,B 0,C 180,E1 -15441.919,E2 -15441.919} C_VEL
LIN {X 0,Y 312.536,Z 545.551,A -85,B 0,C 180,E1 -15444.222,E2 -15444.222} C_VEL
LIN {X 0,Y 312.509,Z 545.558,A -85,B 0,C 180,E1 -15447.335,E2 -15447.335} C_VEL
LIN {X 0,Y 312.557,Z 545.549,A -85,B 0,C 180,E1 -15451.278,E2 -15451.278} C_VEL
LIN {X 0,Y 312.59,Z 545.544,A -85,B 0,C 180,E1 -15454.712,E2 -15454.712} C_VEL
LIN {X 0,Y 312.57,Z 545.552,A -85,B 0,C 180,E1 -15457.528,E2 -15457.528} C_VEL
LIN {X 0,Y 312.588,Z 545.547,A -85,B 0,C 180,E1 -15461.654,E2 -15461.654} C_VEL
LIN {X 0,Y 312.693,Z 545.536,A -85,B 0,C 180,E1 -15465.687,E2 -15465.687} C_VEL
LIN {X 0,Y 312.706,Z 545.535,A -85,B 0,C 180,E1 -15469.643,E2 -15469.643} C_VEL
LIN {X 0,Y 312.86,Z 545.51,A -85,B 0,C 180,E1 -15472.255,E2 -15472.255} C_VEL
LIN {X 0,Y 312.722,Z 545.526,A -85,B 0,C 180,E1 -15474.843,E2 -15474.843} C_VEL
LIN {X 0,Y 312.996,Z 545.494,A -85,B 0,C 180,E1 -15478.714,E2 -15478.714} C_VEL
LIN {X 0,Y 312.996,Z 545.494,A -85,B 0,C 180,E1 -15481.287,E2 -15481.287} C_VEL
LIN {X 0,Y 312.724,Z 545.526,A -85,B 0,C 180,E1 -15485.158,E2 -15485.158} C_VEL
LIN {X 0,Y 312.88,Z 545.512,A -85,B 0,C 180,E1 -15487.746,E2 -15487.746} C_VEL
LIN {X 0,Y 312.677,Z 545.536,A -85,B 0,C 180,E1 -15491.672,E2 -15491.672} C_VEL
LIN {X 0,Y 312.709,Z 545.529,A -85,B 0,C 180,E1 -15494.888,E2 -15494.888} C_VEL
LIN {X 0,Y 312.618,Z 545.541,A -85,B 0,C 180,E1 -15499.225,E2 -15499.225} C_VEL
LIN {X 0,Y 312.534,Z 545.548,A -85,B 0,C 180,E1 -15502.78,E2 -15502.78} C_VEL
LIN {X 0,Y 312.611,Z 545.542,A -85,B 0,C 180,E1 -15505.935,E2 -15505.935} C_VEL
LIN {X 0,Y 312.547,Z 545.551,A -85,B 0,C 180,E1 -15509.65,E2 -15509.65} C_VEL
LIN {X 0,Y 312.528,Z 545.554,A -85,B 0,C 180,E1 -15513.688,E2 -15513.688} C_VEL
LIN {X 0,Y 312.534,Z 545.552,A -85,B 0,C 180,E1 -15517.385,E2 -15517.385} C_VEL
LIN {X 0,Y 312.498,Z 545.558,A -85,B 0,C 180,E1 -15520.709,E2 -15520.709} C_VEL
LIN {X 0,Y 312.46,Z 545.566,A -85,B 0,C 180,E1 -15524.209,E2 -15524.209} C_VEL
LIN {X 0,Y 312.492,Z 545.559,A -85,B 0,C 180,E1 -15527.918,E2 -15527.918} C_VEL
LIN {X 0,Y 312.543,Z 545.552,A -85,B 0,C 180,E1 -15531.909,E2 -15531.909} C_VEL
LIN {X 0,Y 312.514,Z 545.556,A -85,B 0,C 180,E1 -15535.789,E2 -15535.789} C_VEL
LIN {X 0,Y 312.535,Z 545.653,A -85,B 0,C 180,E1 -15537.946,E2 -15537.946} C_VEL
LIN {X 0,Y 315.185,Z 557.858,A -85,B 0,C 180,E1 -15541.715,E2 -15541.715} C_VEL
LIN {X 0,Y 316.805,Z 566.859,A -85,B 0,C 180,E1 -15544.366,E2 -15544.366} C_VEL
LIN {X 0,Y 316.555,Z 570.052,A -85,B 0,C 180,E1 -15545.234,E2 -15545.234} C_VEL
LIN {X 0,Y 322.545,Z 609.968,A -85,B 0,C 180,E1 -15546.678,E2 -15546.678} C_VEL
LIN {X 0,Y 320.813,Z 678.759,A -85,B 0,C 180,E1 -15548.345,E2 -15548.345} C_VEL
LIN {X 0,Y 319.976,Z 692.279,A -85,B 0,C 180,E1 -15548.919,E2 -15548.919} C_VEL
LIN {X 0,Y 318.931,Z 704.63,A -85,B 0,C 180,E1 -15549.69,E2 -15549.69} C_VEL
LIN {X 0,Y 317.809,Z 715.738,A -85,B 0,C 180,E1 -15550.626,E2 -15550.626} C_VEL
LIN {X 0,Y 316.491,Z 727.353,A -85,B 0,C 180,E1 -15551.886,E2 -15551.886} C_VEL
LIN {X 0,Y 315.185,Z 738.043,A -85,B 0,C 180,E1 -15553.347,E2 -15553.347} C_VEL
LIN {X 0,Y 314.214,Z 746.413,A -85,B 0,C 180,E1 -15554.761,E2 -15554.761} C_VEL
LIN {X 0,Y 312.941,Z 755.676,A -85,B 0,C 180,E1 -15556.69,E2 -15556.69} C_VEL
LIN {X 0,Y 311.993,Z 763.124,A -85,B 0,C 180,E1 -15558.631,E2 -15558.631} C_VEL
LIN {X 0,Y 311.454,Z 768.167,A -85,B 0,C 180,E1 -15560.255,E2 -15560.255} C_VEL
LIN {X 0,Y 311.033,Z 773.046,A -85,B 0,C 180,E1 -15562.206,E2 -15562.206} C_VEL
LIN {X 0,Y 310.769,Z 777.013,A -85,B 0,C 180,E1 -15564.304,E2 -15564.304} C_VEL
LIN {X 0,Y 310.727,Z 779.445,A -85,B 0,C 180,E1 -15566.107,E2 -15566.107} C_VEL
LIN {X 0,Y 310.685,Z 780.693,A -85,B 0,C 180,E1 -15567.405,E2 -15567.405} C_VEL
LIN {X 0,Y 310.66,Z 781.515,A -85,B 0,C 180,E1 -15568.702,E2 -15568.702} C_VEL
LIN {X 0,Y 310.692,Z 781.896,A -85,B 0,C 180,E1 -15569.998,E2 -15569.998} C_VEL
LIN {X 0,Y 310.649,Z 781.878,A -85,B 0,C 180,E1 -15571.294,E2 -15571.294} C_VEL
LIN {X 0,Y 310.68,Z 781.469,A -85,B 0,C 180,E1 -15572.591,E2 -15572.591} C_VEL
LIN {X 0,Y 310.704,Z 780.644,A -85,B 0,C 180,E1 -15573.889,E2 -15573.889} C_VEL
LIN {X 0,Y 310.823,Z 777.704,A -85,B 0,C 180,E1 -15576.49,E2 -15576.49} C_VEL
LIN {X 0,Y 311.199,Z 774.359,A -85,B 0,C 180,E1 -15578.439,E2 -15578.439} C_VEL
LIN {X 0,Y 311.756,Z 769.938,A -85,B 0,C 180,E1 -15580.388,E2 -15580.388} C_VEL
LIN {X 0,Y 312.586,Z 764.322,A -85,B 0,C 180,E1 -15582.331,E2 -15582.331} C_VEL
LIN {X 0,Y 313.843,Z 757.331,A -85,B 0,C 180,E1 -15584.258,E2 -15584.258} C_VEL
LIN {X 0,Y 315.242,Z 748.883,A -85,B 0,C 180,E1 -15586.122,E2 -15586.122} C_VEL
LIN {X 0,Y 316.739,Z 739.682,A -85,B 0,C 180,E1 -15587.761,E2 -15587.761} C_VEL
LIN {X 0,Y 318.465,Z 728.761,A -85,B 0,C 180,E1 -15589.329,E2 -15589.329} C_VEL
LIN {X 0,Y 320.081,Z 717.774,A -85,B 0,C 180,E1 -15590.565,E2 -15590.565} C_VEL
LIN {X 0,Y 321.594,Z 705.559,A -85,B 0,C 180,E1 -15591.638,E2 -15591.638} C_VEL
LIN {X 0,Y 322.769,Z 694.12,A -85,B 0,C 180,E1 -15592.396,E2 -15592.396} C_VEL
LIN {X 0,Y 323.77,Z 681.24,A -85,B 0,C 180,E1 -15592.997,E2 -15592.997} C_VEL
LIN {X 0,Y 324.454,Z 666.37,A -85,B 0,C 180,E1 -15593.416,E2 -15593.416} C_VEL
LIN {X 0,Y 326.038,Z 609.288,A -85,B 0,C 180,E1 -15594.815,E2 -15594.815} C_VEL
LIN {X 0,Y 322.865,Z 589.263,A -85,B 0,C 180,E1 -15595.682,E2 -15595.682} C_VEL
LIN {X 0,Y 319.631,Z 573.831,A -85,B 0,C 180,E1 -15596.461,E2 -15596.461} C_VEL
LIN {X 0,Y 317.701,Z 568.699,A -85,B 0,C 180,E1 -15596.849,E2 -15596.849} C_VEL
LIN {X 0,Y 315.925,Z 559.599,A -85,B 0,C 180,E1 -15599.82,E2 -15599.82} C_VEL
LIN {X 0,Y 313.595,Z 549.911,A -85,B 0,C 180,E1 -15603.239,E2 -15603.239} C_VEL
LIN {X 0,Y 312.532,Z 545.556,A -85,B 0,C 180,E1 -15604.889,E2 -15604.889} C_VEL
LIN {X 0,Y 312.553,Z 545.557,A -85,B 0,C 180,E1 -15608.093,E2 -15608.093} C_VEL
LIN {X 0,Y 312.524,Z 545.559,A -85,B 0,C 180,E1 -15612.423,E2 -15612.423} C_VEL
LIN {X 0,Y 312.477,Z 545.565,A -85,B 0,C 180,E1 -15616.028,E2 -15616.028} C_VEL
LIN {X 0,Y 312.494,Z 545.558,A -85,B 0,C 180,E1 -15619.291,E2 -15619.291} C_VEL
LIN {X 0,Y 312.533,Z 545.549,A -85,B 0,C 180,E1 -15622.615,E2 -15622.615} C_VEL
LIN {X 0,Y 312.511,Z 545.552,A -85,B 0,C 180,E1 -15626.309,E2 -15626.309} C_VEL
LIN {X 0,Y 312.537,Z 545.553,A -85,B 0,C 180,E1 -15630.349,E2 -15630.349} C_VEL
LIN {X 0,Y 312.594,Z 545.547,A -85,B 0,C 180,E1 -15634.063,E2 -15634.063} C_VEL
LIN {X 0,Y 312.578,Z 545.545,A -85,B 0,C 180,E1 -15637.528,E2 -15637.528} C_VEL
LIN {X 0,Y 312.628,Z 545.541,A -85,B 0,C 180,E1 -15641.655,E2 -15641.655} C_VEL
LIN {X 0,Y 312.684,Z 545.536,A -85,B 0,C 180,E1 -15645.685,E2 -15645.685} C_VEL
LIN {X 0,Y 312.693,Z 545.536,A -85,B 0,C 180,E1 -15649.641,E2 -15649.641} C_VEL
LIN {X 0,Y 312.861,Z 545.507,A -85,B 0,C 180,E1 -15652.253,E2 -15652.253} C_VEL
LIN {X 0,Y 312.709,Z 545.529,A -85,B 0,C 180,E1 -15654.842,E2 -15654.842} C_VEL
LIN {X 0,Y 312.942,Z 545.505,A -85,B 0,C 180,E1 -15657.425,E2 -15657.425} C_VEL
LIN {X 0,Y 313.11,Z 545.484,A -85,B 0,C 180,E1 -15659.999,E2 -15659.999} C_VEL
LIN {X 0,Y 312.943,Z 545.501,A -85,B 0,C 180,E1 -15662.574,E2 -15662.574} C_VEL
LIN {X 0,Y 312.887,Z 545.509,A -85,B 0,C 180,E1 -15666.62,E2 -15666.62} C_VEL
LIN {X 0,Y 312.776,Z 545.525,A -85,B 0,C 180,E1 -15669.049,E2 -15669.049} C_VEL
LIN {X 0,Y 312.626,Z 545.547,A -85,B 0,C 180,E1 -15672.991,E2 -15672.991} C_VEL
LIN {X 0,Y 312.626,Z 545.546,A -85,B 0,C 180,E1 -15675.65,E2 -15675.65} C_VEL
LIN {X 0,Y 312.637,Z 545.729,A -85,B 0,C 180,E1 -15679.356,E2 -15679.356} C_VEL
LIN {X 0,Y 314.713,Z 554.748,A -85,B 0,C 180,E1 -15682.917,E2 -15682.917} C_VEL
LIN {X 0,Y 323.473,Z 573.864,A -85,B 0,C 180,E1 -15684.423,E2 -15684.423} C_VEL
LIN {X 0,Y 325.447,Z 579.147,A -85,B 0,C 180,E1 -15684.776,E2 -15684.776} C_VEL
LIN {X 0,Y 326.806,Z 586.494,A -85,B 0,C 180,E1 -15685.111,E2 -15685.111} C_VEL
LIN {X 0,Y 324.292,Z 662.054,A -85,B 0,C 180,E1 -15686.972,E2 -15686.972} C_VEL
LIN {X 0,Y 323.453,Z 675.163,A -85,B 0,C 180,E1 -15687.539,E2 -15687.539} C_VEL
LIN {X 0,Y 322.499,Z 686.571,A -85,B 0,C 180,E1 -15688.257,E2 -15688.257} C_VEL
LIN {X 0,Y 321.149,Z 698.527,A -85,B 0,C 180,E1 -15689.254,E2 -15689.254} C_VEL
LIN {X 0,Y 319.812,Z 708.808,A -85,B 0,C 180,E1 -15690.359,E2 -15690.359} C_VEL
LIN {X 0,Y 318.116,Z 720.034,A -85,B 0,C 180,E1 -15691.874,E2 -15691.874} C_VEL
LIN {X 0,Y 316.547,Z 729.381,A -85,B 0,C 180,E1 -15693.45,E2 -15693.45} C_VEL
LIN {X 0,Y 314.892,Z 738.857,A -85,B 0,C 180,E1 -15695.47,E2 -15695.47} C_VEL
LIN {X 0,Y 313.713,Z 745.441,A -85,B 0,C 180,E1 -15697.219,E2 -15697.219} C_VEL
LIN {X 0,Y 312.707,Z 750.875,A -85,B 0,C 180,E1 -15698.997,E2 -15698.997} C_VEL
LIN {X 0,Y 311.817,Z 756.421,A -85,B 0,C 180,E1 -15701.343,E2 -15701.343} C_VEL
LIN {X 0,Y 311.146,Z 760.384,A -85,B 0,C 180,E1 -15703.717,E2 -15703.717} C_VEL
LIN {X 0,Y 310.66,Z 763.124,A -85,B 0,C 180,E1 -15706.379,E2 -15706.379} C_VEL
LIN {X 0,Y 310.417,Z 764.099,A -85,B 0,C 180,E1 -15708.964,E2 -15708.964} C_VEL
LIN {X 0,Y 310.398,Z 763.885,A -85,B 0,C 180,E1 -15710.659,E2 -15710.659} C_VEL
LIN {X 0,Y 310.47,Z 762.957,A -85,B 0,C 180,E1 -15712.398,E2 -15712.398} C_VEL
LIN {X 0,Y 310.729,Z 760.812,A -85,B 0,C 180,E1 -15714.511,E2 -15714.511} C_VEL
LIN {X 0,Y 311.087,Z 757.342,A -85,B 0,C 180,E1 -15716.708,E2 -15716.708} C_VEL
LIN {X 0,Y 311.653,Z 752.331,A -85,B 0,C 180,E1 -15718.972,E2 -15718.972} C_VEL
LIN {X 0,Y 312.297,Z 746.934,A -85,B 0,C 180,E1 -15720.849,E2 -15720.849} C_VEL
LIN {X 0,Y 313.141,Z 740.657,A -85,B 0,C 180,E1 -15722.609,E2 -15722.609} C_VEL
LIN {X 0,Y 314.225,Z 732.344,A -85,B 0,C 180,E1 -15724.5,E2 -15724.5} C_VEL
LIN {X 0,Y 315.421,Z 723.35,A -85,B 0,C 180,E1 -15726.138,E2 -15726.138} C_VEL
LIN {X 0,Y 316.714,Z 712.97,A -85,B 0,C 180,E1 -15727.668,E2 -15727.668} C_VEL
LIN {X 0,Y 317.967,Z 701.498,A -85,B 0,C 180,E1 -15729.015,E2 -15729.015} C_VEL
LIN {X 0,Y 319.138,Z 689.171,A -85,B 0,C 180,E1 -15730.128,E2 -15730.128} C_VEL
LIN {X 0,Y 320.051,Z 677.01,A -85,B 0,C 180,E1 -15730.955,E2 -15730.955} C_VEL
LIN {X 0,Y 320.775,Z 664.789,A -85,B 0,C 180,E1 -15731.541,E2 -15731.541} C_VEL
LIN {X 0,Y 321.233,Z 650.475,A -85,B 0,C 180,E1 -15731.96,E2 -15731.96} C_VEL
LIN {X 0,Y 322.931,Z 584.085,A -85,B 0,C 180,E1 -15733.534,E2 -15733.534} C_VEL
LIN {X 0,Y 319.965,Z 569.677,A -85,B 0,C 180,E1 -15734.105,E2 -15734.105} C_VEL
LIN {X 0,Y 314.202,Z 553.19,A -85,B 0,C 180,E1 -15734.972,E2 -15734.972} C_VEL
LIN {X 0,Y 312.64,Z 545.542,A -85,B 0,C 180,E1 -15737.589,E2 -15737.589} C_VEL
LIN {X 0,Y 312.825,Z 545.518,A -85,B 0,C 180,E1 -15741.303,E2 -15741.303} C_VEL
LIN {X 0,Y 312.899,Z 545.508,A -85,B 0,C 180,E1 -15743.554,E2 -15743.554} C_VEL
LIN {X 0,Y 312.935,Z 545.503,A -85,B 0,C 180,E1 -15747.427,E2 -15747.427} C_VEL
LIN {X 0,Y 313.1,Z 545.481,A -85,B 0,C 180,E1 -15750.002,E2 -15750.002} C_VEL
LIN {X 0,Y 312.935,Z 545.504,A -85,B 0,C 180,E1 -15752.576,E2 -15752.576} C_VEL
LIN {X 0,Y 312.901,Z 545.505,A -85,B 0,C 180,E1 -15756.45,E2 -15756.45} C_VEL
LIN {X 0,Y 312.786,Z 545.526,A -85,B 0,C 180,E1 -15759.051,E2 -15759.051} C_VEL
LIN {X 0,Y 312.634,Z 545.542,A -85,B 0,C 180,E1 -15762.993,E2 -15762.993} C_VEL
LIN {X 0,Y 312.638,Z 545.539,A -85,B 0,C 180,E1 -15765.652,E2 -15765.652} C_VEL
LIN {X 0,Y 312.63,Z 545.542,A -85,B 0,C 180,E1 -15769.238,E2 -15769.238} C_VEL
LIN {X 0,Y 312.546,Z 545.548,A -85,B 0,C 180,E1 -15772.791,E2 -15772.791} C_VEL
LIN {X 0,Y 312.597,Z 545.543,A -85,B 0,C 180,E1 -15775.935,E2 -15775.935} C_VEL
LIN {X 0,Y 312.539,Z 545.552,A -85,B 0,C 180,E1 -15779.652,E2 -15779.652} C_VEL
LIN {X 0,Y 312.521,Z 545.555,A -85,B 0,C 180,E1 -15783.691,E2 -15783.691} C_VEL
LIN {X 0,Y 312.522,Z 545.557,A -85,B 0,C 180,E1 -15787.388,E2 -15787.388} C_VEL
LIN {X 0,Y 312.493,Z 545.556,A -85,B 0,C 180,E1 -15790.711,E2 -15790.711} C_VEL
LIN {X 0,Y 312.475,Z 545.559,A -85,B 0,C 180,E1 -15794.207,E2 -15794.207} C_VEL
LIN {X 0,Y 312.448,Z 545.56,A -85,B 0,C 180,E1 -15795.22,E2 -15795.22} C_VEL
LIN {X 0,Y 311.801,Z 545.644,A -85,B 0,C 180,E1 -15796.296,E2 -15796.296} C_VEL
LIN {X 0,Y 308.951,Z 545.997,A -85,B 0,C 180,E1 -15798.048,E2 -15798.048} C_VEL
LIN {X 0,Y 306.531,Z 546.301,A -85,B 0,C 180,E1 -15799.468,E2 -15799.468} C_VEL
LIN {X 0,Y 305.506,Z 546.424,A -85,B 0,C 180,E1 -15800.568,E2 -15800.568} C_VEL
LIN {X 0,Y 305.43,Z 546.434,A -85,B 0,C 180,E1 -15800.94,E2 -15800.94} C_VEL
LIN {X 0,Y 305.485,Z 546.433,A -85,B 0,C 180,E1 -15803.633,E2 -15803.633} C_VEL
LIN {X 0,Y 305.469,Z 546.431,A -85,B 0,C 180,E1 -15806.485,E2 -15806.485} C_VEL
LIN {X 0,Y 305.501,Z 546.426,A -85,B 0,C 180,E1 -15810.952,E2 -15810.952} C_VEL
LIN {X 0,Y 305.577,Z 546.418,A -85,B 0,C 180,E1 -15814.089,E2 -15814.089} C_VEL
LIN {X 0,Y 305.482,Z 546.43,A -85,B 0,C 180,E1 -15818.402,E2 -15818.402} C_VEL
LIN {X 0,Y 305.549,Z 546.422,A -85,B 0,C 180,E1 -15821.216,E2 -15821.216} C_VEL
LIN {X 0,Y 305.633,Z 546.412,A -85,B 0,C 180,E1 -15825.349,E2 -15825.349} C_VEL
LIN {X 0,Y 305.643,Z 546.412,A -85,B 0,C 180,E1 -15829.401,E2 -15829.401} C_VEL
LIN {X 0,Y 305.804,Z 546.39,A -85,B 0,C 180,E1 -15832.075,E2 -15832.075} C_VEL
LIN {X 0,Y 305.693,Z 546.401,A -85,B 0,C 180,E1 -15834.724,E2 -15834.724} C_VEL
LIN {X 0,Y 305.963,Z 546.37,A -85,B 0,C 180,E1 -15838.684,E2 -15838.684} C_VEL
LIN {X 0,Y 305.963,Z 546.371,A -85,B 0,C 180,E1 -15841.317,E2 -15841.317} C_VEL
LIN {X 0,Y 305.861,Z 546.383,A -85,B 0,C 180,E1 -15846.598,E2 -15846.598} C_VEL
LIN {X 0,Y 305.744,Z 546.398,A -85,B 0,C 180,E1 -15849.26,E2 -15849.26} C_VEL
LIN {X 0,Y 305.597,Z 546.414,A -85,B 0,C 180,E1 -15853.296,E2 -15853.296} C_VEL
LIN {X 0,Y 305.602,Z 546.421,A -85,B 0,C 180,E1 -15856.02,E2 -15856.02} C_VEL
LIN {X 0,Y 305.569,Z 546.42,A -85,B 0,C 180,E1 -15859.436,E2 -15859.436} C_VEL
LIN {X 0,Y 305.495,Z 546.423,A -85,B 0,C 180,E1 -15863.039,E2 -15863.039} C_VEL
LIN {X 0,Y 305.555,Z 546.423,A -85,B 0,C 180,E1 -15866.227,E2 -15866.227} C_VEL
LIN {X 0,Y 305.496,Z 546.428,A -85,B 0,C 180,E1 -15869.047,E2 -15869.047} C_VEL
LIN {X 0,Y 305.451,Z 546.437,A -85,B 0,C 180,E1 -15871.952,E2 -15871.952} C_VEL
LIN {X 0,Y 305.471,Z 546.431,A -85,B 0,C 180,E1 -15875.113,E2 -15875.113} C_VEL
LIN {X 0,Y 305.475,Z 546.434,A -85,B 0,C 180,E1 -15878.532,E2 -15878.532} C_VEL
LIN {X 0,Y 305.463,Z 546.435,A -85,B 0,C 180,E1 -15882.585,E2 -15882.585} C_VEL
LIN {X 0,Y 305.433,Z 546.44,A -85,B 0,C 180,E1 -15886.344,E2 -15886.344} C_VEL
LIN {X 0,Y 305.466,Z 546.433,A -85,B 0,C 180,E1 -15889.892,E2 -15889.892} C_VEL
LIN {X 0,Y 305.507,Z 546.428,A -85,B 0,C 180,E1 -15893.626,E2 -15893.626} C_VEL
